C09159=1159.739,-99.599,-42.687,178.880,5.876,149.381
C09160=1159.744,-99.849,-42.678,178.877,5.876,149.382
C09161=1159.750,-100.100,-42.669,178.875,5.875,149.382
C09162=1159.755,-100.349,-42.659,178.874,5.875,149.383
C09163=1159.760,-100.599,-42.650,178.871,5.875,149.383
C09164=1159.766,-100.849,-42.641,178.869,5.875,149.384
C09165=1159.771,-101.098,-42.631,178.867,5.874,149.384
C09166=1159.777,-101.348,-42.622,178.864,5.874,149.385
C09167=1159.782,-101.598,-42.613,178.863,5.874,149.386
C09168=1159.787,-101.848,-42.604,178.861,5.873,149.386
C09169=1159.793,-102.120,-42.594,178.859,5.874,149.387
C09170=1159.799,-102.392,-42.583,178.856,5.873,149.387
C09171=1159.805,-102.664,-42.573,178.854,5.872,149.388
C09172=1159.810,-102.936,-42.562,178.852,5.872,149.389
C09173=1159.815,-103.186,-42.554,178.849,5.872,149.389
C09174=1159.821,-103.436,-42.544,178.847,5.871,149.390
C09175=1159.826,-103.686,-42.535,178.846,5.871,149.390
C09176=1159.831,-103.935,-42.526,178.843,5.871,149.391
C09177=1159.836,-104.185,-42.517,178.841,5.870,149.391
C09178=1159.842,-104.435,-42.507,178.839,5.870,149.392
C09179=1159.847,-104.685,-42.498,178.837,5.870,149.393
C09180=1159.853,-104.933,-42.489,178.835,5.870,149.393
C09181=1159.859,-105.184,-42.479,178.833,5.869,149.394
C09182=1159.864,-105.433,-42.471,178.831,5.870,149.394
C09183=1159.869,-105.683,-42.462,178.828,5.869,149.395
C09184=1159.874,-105.933,-42.453,178.826,5.868,149.395
C09185=1159.880,-106.183,-42.443,178.825,5.868,149.396
C09186=1159.885,-106.432,-42.434,178.822,5.868,149.396
C09187=1159.890,-106.682,-42.425,178.820,5.868,149.397
C09188=1159.895,-106.932,-42.416,178.818,5.867,149.397
C09189=1159.901,-107.182,-42.406,178.816,5.867,149.398
C09190=1159.906,-107.432,-42.397,178.814,5.867,149.399
C09191=1159.911,-107.681,-42.388,178.812,5.866,149.399
C09192=1159.917,-107.931,-42.379,178.810,5.866,149.400
C09193=1159.922,-108.181,-42.369,178.807,5.865,149.400
C09194=1159.928,-108.431,-42.361,178.806,5.865,149.401
C09195=1159.933,-108.680,-42.352,178.804,5.865,149.401
C09196=1159.939,-108.930,-42.343,178.802,5.865,149.402
C09197=1159.944,-109.180,-42.334,178.799,5.864,149.403
C09198=1159.949,-109.430,-42.324,178.797,5.864,149.403
C09199=1159.954,-109.680,-42.315,178.795,5.864,149.404
C09200=1159.960,-109.929,-42.306,178.793,5.863,149.404
C09201=1159.965,-110.179,-42.297,178.791,5.863,149.405
C09202=1159.970,-110.429,-42.288,178.789,5.863,149.405
C09203=1159.976,-110.679,-42.279,178.787,5.863,149.406
C09204=1159.982,-110.928,-42.270,178.785,5.862,149.406
C09205=1159.987,-111.178,-42.262,178.783,5.862,149.407
C09206=1159.992,-111.428,-42.253,178.781,5.862,149.408
C09207=1159.997,-111.678,-42.244,178.778,5.861,149.408
C09208=1160.002,-111.928,-42.235,178.777,5.861,149.409
C09209=1160.008,-112.178,-42.225,178.775,5.860,149.409
C09210=1160.013,-112.428,-42.216,178.773,5.861,149.410
C09211=1160.019,-112.678,-42.208,178.770,5.860,149.410
C09212=1160.024,-112.927,-42.199,178.769,5.860,149.411
C09213=1160.029,-113.177,-42.190,178.767,5.859,149.411
C09214=1160.035,-113.427,-42.181,178.764,5.860,149.412
C09215=1160.040,-113.676,-42.172,178.762,5.859,149.412
C09216=1160.045,-113.926,-42.163,178.761,5.859,149.413
C09217=1160.051,-114.176,-42.154,178.758,5.858,149.413
C09218=1160.057,-114.426,-42.145,178.756,5.858,149.414
C09219=1160.062,-114.675,-42.137,178.754,5.858,149.415
C09220=1160.067,-114.925,-42.128,178.752,5.857,149.415
C09221=1160.072,-115.175,-42.119,178.750,5.857,149.416
C09222=1160.077,-115.425,-42.110,178.748,5.857,149.416
C09223=1160.082,-115.675,-42.101,178.746,5.857,149.417
C09224=1160.088,-115.924,-42.092,178.744,5.856,149.417
C09225=1160.093,-116.174,-42.083,178.742,5.857,149.418
C09226=1160.099,-116.424,-42.075,178.740,5.856,149.418
C09227=1160.104,-116.674,-42.065,178.738,5.856,149.419
C09228=1160.110,-116.924,-42.056,178.736,5.855,149.419
C09229=1160.115,-117.173,-42.048,178.734,5.855,149.420
C09230=1160.121,-117.423,-42.039,178.732,5.855,149.421
C09231=1160.126,-117.673,-42.031,178.730,5.855,149.421
C09232=1160.131,-117.923,-42.022,178.728,5.854,149.422
C09233=1160.136,-118.173,-42.013,178.726,5.853,149.422
C09234=1160.142,-118.422,-42.004,178.724,5.854,149.423
C09235=1160.147,-118.672,-41.995,178.721,5.853,149.423
C09236=1160.152,-118.922,-41.986,178.720,5.853,149.424
C09237=1160.158,-119.172,-41.978,178.718,5.852,149.424
C09238=1160.164,-119.421,-41.970,178.715,5.853,149.425
C09239=1160.169,-119.671,-41.961,178.713,5.852,149.425
C09240=1160.174,-119.921,-41.952,178.712,5.852,149.426
C09241=1160.179,-120.171,-41.943,178.709,5.851,149.426
C09242=1160.185,-120.420,-41.935,178.707,5.852,149.427
C09243=1160.190,-120.670,-41.926,178.705,5.851,149.428
C09244=1160.196,-120.920,-41.917,178.704,5.851,149.428
C09245=1160.201,-121.170,-41.909,178.701,5.850,149.429
C09246=1160.207,-121.419,-41.900,178.699,5.851,149.429
C09247=1160.212,-121.669,-41.891,178.697,5.850,149.430
C09248=1160.217,-121.919,-41.882,178.696,5.850,149.430
C09249=1160.222,-122.169,-41.874,178.693,5.849,149.431
C09250=1160.228,-122.419,-41.866,178.692,5.849,149.431
C09251=1160.233,-122.668,-41.857,178.689,5.849,149.432
C09252=1160.238,-122.918,-41.848,178.687,5.849,149.432
C09253=1160.244,-123.169,-41.840,178.685,5.848,149.433
C09254=1160.250,-123.418,-41.831,178.684,5.848,149.433
C09255=1160.254,-123.668,-41.823,178.681,5.847,149.434
C09256=1160.259,-123.917,-41.814,178.679,5.848,149.435
C09257=1160.265,-124.168,-41.806,178.677,5.847,149.435
C09258=1160.271,-124.417,-41.797,178.676,5.847,149.436
C09259=1160.276,-124.667,-41.788,178.673,5.846,149.436
C09260=1160.281,-124.917,-41.780,178.671,5.847,149.437
C09261=1160.287,-125.166,-41.771,178.669,5.846,149.437
C09262=1160.292,-125.416,-41.763,178.668,5.846,149.438
C09263=1160.297,-125.666,-41.754,178.665,5.845,149.438
C09264=1160.303,-125.916,-41.746,178.664,5.845,149.439
C09265=1160.309,-126.166,-41.737,178.661,5.845,149.439
C09266=1160.313,-126.415,-41.729,178.659,5.845,149.440
C09267=1160.319,-126.665,-41.721,178.657,5.844,149.440
C09268=1160.324,-126.915,-41.712,178.656,5.844,149.441
C09269=1160.329,-127.165,-41.703,178.653,5.843,149.441
C09270=1160.335,-127.415,-41.695,178.651,5.844,149.442
C09271=1160.341,-127.664,-41.686,178.649,5.843,149.443
C09272=1160.346,-127.915,-41.678,178.648,5.843,149.443
C09273=1159.925,-127.926,-41.720,178.644,5.846,149.445
C09274=1159.919,-127.675,-41.728,178.645,5.846,149.444
C09275=1159.914,-127.425,-41.737,178.648,5.847,149.444
C09276=1159.908,-127.176,-41.745,178.650,5.847,149.443
C09277=1159.903,-126.926,-41.753,178.652,5.847,149.443
C09278=1159.898,-126.676,-41.762,178.653,5.847,149.442
C09279=1159.892,-126.427,-41.771,178.656,5.848,149.442
C09280=1159.887,-126.177,-41.779,178.658,5.848,149.441
C09281=1159.882,-125.927,-41.788,178.660,5.848,149.441
C09282=1159.876,-125.678,-41.796,178.661,5.848,149.440
C09283=1159.871,-125.427,-41.804,178.664,5.849,149.440
C09284=1159.865,-125.177,-41.813,178.665,5.849,149.439
C09285=1159.860,-124.927,-41.822,178.668,5.849,149.438
C09286=1159.855,-124.679,-41.830,178.670,5.849,149.438
C09287=1159.850,-124.428,-41.838,178.672,5.850,149.437
C09288=1159.845,-124.178,-41.847,178.673,5.850,149.437
C09289=1159.839,-123.929,-41.856,178.676,5.851,149.436
C09290=1159.833,-123.679,-41.864,178.678,5.851,149.436
C09291=1159.828,-123.429,-41.873,178.680,5.851,149.435
C09292=1159.822,-123.180,-41.881,178.681,5.851,149.435
C09293=1159.817,-122.930,-41.890,178.684,5.852,149.434
C09294=1159.812,-122.679,-41.898,178.685,5.852,149.434
C09295=1159.807,-122.430,-41.907,178.688,5.852,149.433
C09296=1159.801,-122.180,-41.916,178.690,5.853,149.433
C09297=1159.796,-121.931,-41.925,178.692,5.853,149.432
C09298=1159.790,-121.680,-41.933,178.694,5.854,149.432
C09299=1159.785,-121.430,-41.942,178.696,5.853,149.431
C09300=1159.779,-121.181,-41.950,178.698,5.854,149.430
C09301=1159.774,-120.931,-41.959,178.700,5.854,149.430
C09302=1159.769,-120.681,-41.968,178.702,5.855,149.429
C09303=1159.764,-120.432,-41.977,178.704,5.855,149.429
C09304=1159.758,-120.182,-41.985,178.706,5.855,149.428
C09305=1159.752,-119.932,-41.994,178.708,5.855,149.428
C09306=1159.747,-119.682,-42.003,178.710,5.856,149.427
C09307=1159.742,-119.432,-42.011,178.712,5.856,149.427
C09308=1159.736,-119.183,-42.020,178.714,5.856,149.426
C09309=1159.731,-118.933,-42.029,178.716,5.856,149.426
C09310=1159.726,-118.683,-42.037,178.718,5.857,149.425
C09311=1159.721,-118.433,-42.046,178.720,5.857,149.425
C09312=1159.715,-118.183,-42.055,178.722,5.858,149.424
C09313=1159.710,-117.934,-42.063,178.724,5.857,149.423
C09314=1159.704,-117.684,-42.072,178.726,5.858,149.423
C09315=1159.699,-117.434,-42.081,178.728,5.858,149.422
C09316=1159.694,-117.184,-42.090,178.730,5.859,149.422
C09317=1159.689,-116.934,-42.099,178.732,5.858,149.421
C09318=1159.683,-116.685,-42.107,178.734,5.859,149.421
C09319=1159.678,-116.435,-42.116,178.736,5.860,149.420
C09320=1159.673,-116.185,-42.125,178.738,5.860,149.420
C09321=1159.667,-115.935,-42.134,178.741,5.860,149.419
C09322=1159.662,-115.685,-42.142,178.742,5.860,149.419
C09323=1159.656,-115.436,-42.151,178.744,5.861,149.418
C09324=1159.651,-115.186,-42.160,178.746,5.861,149.418
C09325=1159.645,-114.936,-42.169,178.749,5.861,149.417
C09326=1159.640,-114.686,-42.178,178.750,5.861,149.416
C09327=1159.635,-114.436,-42.187,178.753,5.862,149.416
C09328=1159.629,-114.187,-42.196,178.754,5.862,149.415
C09329=1159.624,-113.937,-42.205,178.757,5.862,149.415
C09330=1159.619,-113.688,-42.213,178.758,5.862,149.414
C09331=1159.614,-113.438,-42.222,178.761,5.863,149.414
C09332=1159.609,-113.188,-42.231,178.763,5.864,149.413
C09333=1159.603,-112.938,-42.241,178.765,5.863,149.413
C09334=1159.597,-112.689,-42.249,178.767,5.864,149.412
C09335=1159.592,-112.439,-42.258,178.769,5.864,149.412
C09336=1159.587,-112.189,-42.267,178.771,5.864,149.411
C09337=1159.581,-111.939,-42.276,178.773,5.864,149.410
C09338=1159.576,-111.689,-42.285,178.775,5.865,149.410
C09339=1159.571,-111.439,-42.294,178.777,5.865,149.409
C09340=1159.565,-111.189,-42.303,178.779,5.865,149.409
C09341=1159.560,-110.939,-42.312,178.781,5.865,149.408
C09342=1159.554,-110.690,-42.321,178.783,5.866,149.408
C09343=1159.549,-110.440,-42.330,178.785,5.867,149.407
C09344=1159.544,-110.190,-42.339,178.787,5.867,149.407
C09345=1159.539,-109.941,-42.347,178.790,5.867,149.406
C09346=1159.533,-109.690,-42.357,178.791,5.867,149.406
C09347=1159.528,-109.441,-42.366,178.794,5.868,149.405
C09348=1159.523,-109.191,-42.375,178.796,5.868,149.404
C09349=1159.518,-108.941,-42.384,178.798,5.868,149.404
C09350=1159.513,-108.692,-42.393,178.799,5.868,149.403
C09351=1159.506,-108.442,-42.402,178.802,5.869,149.403
C09352=1159.501,-108.192,-42.411,178.804,5.869,149.402
C09353=1159.496,-107.942,-42.420,178.806,5.869,149.402
C09354=1159.491,-107.693,-42.429,178.808,5.870,149.401
C09355=1159.485,-107.442,-42.439,178.810,5.870,149.400
C09356=1159.480,-107.193,-42.448,178.812,5.871,149.400
C09357=1159.475,-106.943,-42.457,178.814,5.871,149.400
C09358=1159.469,-106.694,-42.466,178.817,5.871,149.399
C09359=1159.464,-106.443,-42.475,178.819,5.872,149.398
C09360=1159.458,-106.193,-42.484,178.820,5.872,149.398
C09361=1159.453,-105.944,-42.493,178.823,5.872,149.397
C09362=1159.448,-105.694,-42.503,178.825,5.872,149.397
C09363=1159.442,-105.444,-42.512,178.827,5.873,149.396
C09364=1159.437,-105.195,-42.521,178.829,5.872,149.395
C09365=1159.432,-104.945,-42.530,178.831,5.873,149.395
C09366=1159.426,-104.695,-42.539,178.833,5.874,149.394
C09367=1159.421,-104.446,-42.549,178.835,5.874,149.394
C09368=1159.416,-104.196,-42.558,178.838,5.874,149.393
C09369=1159.410,-103.946,-42.567,178.839,5.874,149.393
C09370=1159.405,-103.696,-42.576,178.841,5.875,149.392
C09371=1159.400,-103.447,-42.586,178.844,5.875,149.392
C09372=1159.394,-103.197,-42.595,178.846,5.875,149.391
C09373=1159.389,-102.947,-42.604,178.848,5.876,149.391
C09374=1159.383,-102.675,-42.614,178.850,5.876,149.390
C09375=1159.378,-102.403,-42.625,178.852,5.876,149.389
C09376=1159.372,-102.131,-42.635,178.855,5.877,149.389
C09377=1159.366,-101.859,-42.644,178.857,5.878,149.388
C09378=1159.361,-101.610,-42.654,178.859,5.877,149.387
C09379=1159.355,-101.360,-42.663,178.861,5.878,149.387
C09380=1159.350,-101.110,-42.672,178.863,5.878,149.387
C09381=1159.345,-100.861,-42.682,178.866,5.878,149.386
C09382=1159.339,-100.610,-42.691,178.868,5.879,149.385
C09383=1159.334,-100.360,-42.700,178.869,5.879,149.385
C09384=1159.329,-100.110,-42.711,178.872,5.879,149.384
C09385=1159.324,-99.861,-42.719,178.874,5.879,149.384
C09386=1159.318,-99.611,-42.728,178.876,5.880,149.383
C09387=1159.313,-99.361,-42.739,178.878,5.880,149.382
C09388=1159.308,-99.111,-42.747,178.880,5.880,149.382
C09389=1159.302,-98.861,-42.757,178.882,5.881,149.381
C09390=1159.297,-98.612,-42.767,178.884,5.881,149.381
C09391=1159.292,-98.362,-42.775,178.886,5.882,149.380
C09392=1159.286,-98.113,-42.786,178.889,5.882,149.380
C09393=1159.281,-97.863,-42.795,178.891,5.882,149.379
C09394=1159.275,-97.612,-42.804,178.893,5.883,149.379
C09395=1159.270,-97.363,-42.814,178.895,5.883,149.378
C09396=1159.265,-97.113,-42.823,178.897,5.883,149.377
C09397=1159.260,-96.864,-42.833,178.899,5.884,149.377
C09398=1159.254,-96.614,-42.842,178.901,5.884,149.376
C09399=1159.248,-96.364,-42.851,178.904,5.884,149.376
C09400=1159.244,-96.115,-42.861,178.905,5.884,149.375
C09401=1159.238,-95.864,-42.870,178.907,5.885,149.375
C09402=1159.233,-95.615,-42.880,178.910,5.885,149.374
C09403=1159.227,-95.365,-42.889,178.912,5.885,149.374
C09404=1159.222,-95.116,-42.899,178.914,5.886,149.373
C09405=1159.216,-94.866,-42.909,178.917,5.886,149.372
C09406=1159.212,-94.616,-42.918,178.918,5.886,149.372
C09407=1159.206,-94.366,-42.928,178.920,5.887,149.371
C09408=1159.201,-94.116,-42.938,178.922,5.887,149.371
C09409=1159.195,-93.866,-42.947,178.925,5.887,149.370
C09410=1159.190,-93.617,-42.957,178.927,5.888,149.370
C09411=1159.184,-93.367,-42.966,178.929,5.888,149.369
C09412=1159.180,-93.118,-42.976,178.931,5.889,149.369
C09413=1159.174,-92.867,-42.985,178.933,5.889,149.368
C09414=1159.169,-92.618,-42.995,178.935,5.889,149.367
C09415=1159.163,-92.368,-43.004,178.938,5.890,149.367
C09416=1159.159,-92.118,-43.014,178.940,5.889,149.366
C09417=1159.153,-91.868,-43.024,178.942,5.890,149.366
C09418=1159.148,-91.619,-43.033,178.944,5.891,149.365
C09419=1159.142,-91.369,-43.044,178.946,5.890,149.364
C09420=1159.137,-91.119,-43.053,178.948,5.891,149.364
C09421=1159.132,-90.870,-43.063,178.951,5.892,149.363
C09422=1159.126,-90.620,-43.072,178.953,5.892,149.363
C09423=1159.121,-90.370,-43.082,178.955,5.892,149.362
C09424=1159.116,-90.120,-43.091,178.957,5.893,149.362
C09425=1159.111,-89.870,-43.101,178.959,5.893,149.361
C09426=1159.105,-89.621,-43.112,178.961,5.893,149.361
C09427=1159.100,-89.371,-43.120,178.963,5.893,149.360
C09428=1159.094,-89.121,-43.131,178.966,5.894,149.359
C09429=1159.089,-88.872,-43.140,178.968,5.895,149.359
C09430=1159.084,-88.621,-43.150,178.970,5.894,149.358
C09431=1159.078,-88.372,-43.160,178.972,5.895,149.358
C09432=1159.074,-88.122,-43.170,178.974,5.896,149.357
C09433=1159.068,-87.872,-43.179,178.976,5.895,149.357
C09434=1159.063,-87.623,-43.189,178.978,5.896,149.356
C09435=1159.057,-87.374,-43.199,178.981,5.897,149.356
C09436=1159.052,-87.123,-43.209,178.983,5.896,149.355
C09437=1159.047,-86.873,-43.219,178.985,5.897,149.354
C09438=1159.041,-86.624,-43.229,178.988,5.898,149.354
C09439=1159.036,-86.374,-43.238,178.989,5.898,149.353
C09440=1159.031,-86.124,-43.248,178.991,5.898,149.353
C09441=1159.026,-85.874,-43.259,178.994,5.899,149.352
C09442=1159.021,-85.625,-43.268,178.996,5.899,149.352
C09443=1159.015,-85.375,-43.278,178.998,5.899,149.351
C09444=1159.009,-85.125,-43.288,179.001,5.900,149.350
C09445=1159.005,-84.875,-43.298,179.002,5.900,149.350
C09446=1159.000,-84.626,-43.308,179.005,5.900,149.349
C09447=1158.994,-84.376,-43.318,179.007,5.901,149.349
C09448=1158.989,-84.126,-43.327,179.009,5.901,149.348
C09449=1158.983,-83.877,-43.337,179.011,5.901,149.347
C09450=1158.978,-83.627,-43.348,179.013,5.902,149.347
C09451=1158.973,-83.377,-43.357,179.016,5.902,149.346
C09452=1158.967,-83.127,-43.367,179.018,5.902,149.346
C09453=1158.962,-82.878,-43.377,179.020,5.903,149.345
C09454=1158.957,-82.627,-43.388,179.022,5.903,149.345
C09455=1158.952,-82.378,-43.398,179.024,5.904,149.344
C09456=1158.946,-82.128,-43.407,179.027,5.904,149.343
C09457=1158.940,-81.879,-43.417,179.028,5.904,149.343
C09458=1158.936,-81.629,-43.427,179.031,5.905,149.342
C09459=1158.931,-81.379,-43.437,179.033,5.905,149.342
C09460=1158.925,-81.129,-43.448,179.035,5.905,149.341
C09461=1158.919,-80.880,-43.458,179.038,5.906,149.341
C09462=1158.915,-80.630,-43.468,179.040,5.906,149.340
C09463=1158.909,-80.380,-43.477,179.041,5.906,149.340
C09464=1158.904,-80.130,-43.488,179.044,5.907,149.339
C09465=1158.899,-79.880,-43.498,179.046,5.907,149.338
C09466=1158.893,-79.631,-43.508,179.048,5.907,149.338
C09467=1158.888,-79.381,-43.518,179.050,5.908,149.337
C09468=1158.883,-79.132,-43.528,179.053,5.909,149.337
C09469=1158.878,-78.881,-43.539,179.055,5.909,149.336
C09470=1158.872,-78.632,-43.549,179.057,5.909,149.336
C09471=1158.867,-78.383,-43.559,179.060,5.909,149.335
C09472=1158.862,-78.132,-43.569,179.062,5.910,149.334
C09473=1158.857,-77.883,-43.579,179.063,5.910,149.334
C09474=1158.851,-77.633,-43.589,179.066,5.910,149.333
C09475=1158.845,-77.383,-43.599,179.068,5.911,149.333
C09476=1158.840,-77.133,-43.610,179.070,5.911,149.332
C09477=1158.835,-76.884,-43.619,179.073,5.912,149.331
C09478=1158.829,-76.612,-43.631,179.075,5.912,149.331
C09479=1158.823,-76.342,-43.641,179.077,5.913,149.330
C09480=1158.818,-76.070,-43.653,179.080,5.913,149.330
C09481=1158.812,-75.798,-43.664,179.082,5.913,149.329
C09482=1158.807,-75.549,-43.674,179.084,5.914,149.328
C09483=1158.802,-75.299,-43.685,179.087,5.914,149.328
C09484=1158.796,-75.049,-43.695,179.089,5.915,149.327
C09485=1158.791,-74.800,-43.705,179.091,5.915,149.327
C09486=1158.786,-74.550,-43.716,179.093,5.915,149.326
C09487=1158.780,-74.300,-43.726,179.096,5.916,149.325
C09488=1158.774,-74.050,-43.736,179.097,5.916,149.325
C09489=1158.770,-73.801,-43.747,179.100,5.916,149.324
C09490=1158.765,-73.552,-43.757,179.102,5.917,149.324
C09491=1158.759,-73.302,-43.767,179.105,5.917,149.323
C09492=1158.754,-73.052,-43.778,179.106,5.917,149.323
C09493=1158.749,-72.802,-43.788,179.109,5.918,149.322
C09494=1158.743,-72.553,-43.798,179.111,5.919,149.321
C09495=1158.738,-72.302,-43.809,179.113,5.919,149.321
C09496=1158.732,-72.053,-43.819,179.115,5.919,149.320
C09497=1158.727,-71.803,-43.829,179.118,5.920,149.320
C09498=1158.722,-71.553,-43.840,179.120,5.920,149.319
C09499=1158.716,-71.304,-43.850,179.122,5.920,149.319
C09500=1158.712,-71.054,-43.861,179.125,5.920,149.318
C09501=1158.706,-70.804,-43.871,179.127,5.921,149.317
C09502=1158.701,-70.554,-43.882,179.129,5.922,149.317
C09503=1158.695,-70.305,-43.892,179.131,5.922,149.316
C09504=1158.690,-70.055,-43.902,179.133,5.922,149.316
C09505=1158.685,-69.805,-43.913,179.136,5.923,149.315
C09506=1158.679,-69.556,-43.924,179.138,5.923,149.315
C09507=1158.674,-69.306,-43.934,179.140,5.923,149.314
C09508=1158.669,-69.056,-43.945,179.142,5.924,149.313
C09509=1158.664,-68.806,-43.955,179.145,5.925,149.313
C09510=1158.658,-68.556,-43.965,179.147,5.924,149.312
C09511=1158.653,-68.307,-43.976,179.149,5.925,149.312
C09512=1158.648,-68.057,-43.987,179.152,5.926,149.311
C09513=1158.642,-67.808,-43.997,179.154,5.926,149.310
C09514=1158.637,-67.557,-44.008,179.156,5.926,149.310
C09515=1158.632,-67.308,-44.018,179.158,5.927,149.309
C09516=1158.627,-67.058,-44.029,179.161,5.927,149.309
C09517=1158.621,-66.809,-44.039,179.163,5.928,149.308
C09518=1158.616,-66.558,-44.050,179.164,5.928,149.308
C09519=1158.611,-66.310,-44.061,179.167,5.928,149.307
C09520=1158.606,-66.059,-44.072,179.169,5.929,149.306
C09521=1158.601,-65.810,-44.082,179.172,5.929,149.306
C09522=1158.596,-65.559,-44.092,179.174,5.929,149.305
C09523=1158.590,-65.311,-44.103,179.176,5.930,149.305
C09524=1158.585,-65.060,-44.114,179.178,5.931,149.304
C09525=1158.580,-64.811,-44.124,179.181,5.931,149.303
C09526=1158.575,-64.561,-44.135,179.183,5.931,149.303
C09527=1158.569,-64.312,-44.145,179.185,5.932,149.302
C09528=1158.564,-64.061,-44.156,179.188,5.932,149.302
C09529=1158.558,-63.812,-44.168,179.190,5.933,149.301
C09530=1158.553,-63.562,-44.178,179.192,5.933,149.301
C09531=1158.548,-63.312,-44.188,179.194,5.933,149.300
C09532=1158.543,-63.063,-44.200,179.197,5.934,149.299
C09533=1158.537,-62.813,-44.210,179.199,5.935,149.299
C09534=1158.532,-62.563,-44.220,179.201,5.935,149.298
C09535=1158.527,-62.314,-44.231,179.203,5.935,149.298
C09536=1158.522,-62.064,-44.242,179.206,5.935,149.297
C09537=1158.516,-61.815,-44.253,179.208,5.936,149.296
C09538=1158.511,-61.564,-44.264,179.210,5.937,149.296
C09539=1158.506,-61.315,-44.275,179.212,5.937,149.295
C09540=1158.501,-61.065,-44.286,179.214,5.937,149.295
C09541=1158.495,-60.816,-44.296,179.217,5.938,149.294
C09542=1158.491,-60.566,-44.307,179.219,5.938,149.294
C09543=1158.486,-60.316,-44.318,179.221,5.938,149.293
C09544=1158.480,-60.066,-44.329,179.223,5.939,149.292
C09545=1158.475,-59.816,-44.340,179.226,5.939,149.292
C09546=1158.469,-59.567,-44.351,179.228,5.940,149.291
C09547=1158.464,-59.317,-44.361,179.231,5.940,149.291
C09548=1158.459,-59.068,-44.372,179.233,5.940,149.290
C09549=1158.453,-58.818,-44.383,179.235,5.941,149.289
C09550=1158.449,-58.568,-44.395,179.237,5.942,149.289
C09551=1158.443,-58.318,-44.405,179.240,5.942,149.288
C09552=1158.438,-58.069,-44.416,179.242,5.943,149.288
C09553=1158.433,-57.819,-44.426,179.244,5.943,149.287
C09554=1158.427,-57.569,-44.438,179.247,5.943,149.287
C09555=1158.422,-57.319,-44.449,179.249,5.944,149.286
C09556=1158.417,-57.070,-44.460,179.251,5.944,149.285
C09557=1158.412,-56.820,-44.470,179.254,5.945,149.285
C09558=1158.406,-56.571,-44.482,179.256,5.945,149.284
C09559=1158.401,-56.320,-44.492,179.258,5.946,149.284
C09560=1158.396,-56.071,-44.504,179.261,5.946,149.283
C09561=1158.391,-55.822,-44.515,179.263,5.947,149.283
C09562=1158.385,-55.571,-44.526,179.265,5.947,149.282
C09563=1158.380,-55.322,-44.537,179.267,5.947,149.281
C09564=1158.375,-55.072,-44.547,179.270,5.948,149.281
C09565=1158.370,-54.822,-44.559,179.272,5.948,149.280
C09566=1158.364,-54.573,-44.570,179.274,5.949,149.280
C09567=1158.359,-54.323,-44.581,179.277,5.950,149.279
C09568=1158.354,-54.073,-44.592,179.278,5.950,149.279
C09569=1158.349,-53.824,-44.603,179.281,5.950,149.278
C09570=1158.343,-53.574,-44.614,179.283,5.951,149.277
C09571=1158.339,-53.324,-44.625,179.286,5.951,149.277
C09572=1158.333,-53.075,-44.635,179.288,5.952,149.276
C09573=1158.328,-52.825,-44.647,179.290,5.952,149.275
C09574=1158.323,-52.575,-44.659,179.292,5.952,149.275
C09575=1158.317,-52.326,-44.669,179.295,5.953,149.274
C09576=1158.312,-52.076,-44.681,179.297,5.954,149.274
C09577=1158.307,-51.826,-44.692,179.300,5.954,149.273
C09578=1158.302,-51.577,-44.703,179.302,5.955,149.273
C09579=1158.296,-51.327,-44.714,179.304,5.954,149.272
C09580=1158.292,-51.077,-44.725,179.306,5.955,149.271
C09581=1158.286,-50.828,-44.737,179.309,5.956,149.271
C09582=1158.281,-50.557,-44.749,179.311,5.956,149.270
C09583=1158.275,-50.286,-44.761,179.314,5.957,149.270
C09584=1158.269,-50.016,-44.773,179.316,5.957,149.269
C09585=1158.264,-49.745,-44.786,179.319,5.958,149.268
C09586=1158.259,-49.495,-44.796,179.321,5.958,149.268
C09587=1158.253,-49.246,-44.808,179.323,5.959,149.267
C09588=1158.248,-48.996,-44.819,179.326,5.959,149.266
C09589=1158.242,-48.746,-44.831,179.328,5.960,149.266
C09590=1158.237,-48.496,-44.842,179.330,5.960,149.265
C09591=1158.231,-48.247,-44.853,179.333,5.961,149.265
C09592=1158.227,-47.997,-44.864,179.335,5.961,149.264
C09593=1158.222,-47.748,-44.876,179.337,5.962,149.264
C09594=1158.216,-47.498,-44.887,179.340,5.962,149.263
C09595=1158.211,-47.249,-44.898,179.342,5.962,149.262
C09596=1158.206,-46.998,-44.910,179.344,5.963,149.262
C09597=1158.201,-46.749,-44.921,179.347,5.964,149.261
C09598=1158.195,-46.499,-44.932,179.349,5.964,149.261
C09599=1158.190,-46.250,-44.944,179.351,5.965,149.260
C09600=1158.185,-46.000,-44.956,179.354,5.965,149.259
C09601=1158.180,-45.750,-44.967,179.356,5.965,149.259
C09602=1158.174,-45.501,-44.978,179.358,5.966,149.258
C09603=1158.169,-45.251,-44.989,179.360,5.966,149.258
C09604=1158.164,-45.001,-45.001,179.363,5.967,149.257
C09605=1158.159,-44.751,-45.012,179.365,5.968,149.257
C09606=1158.153,-44.501,-45.024,179.368,5.968,149.256
C09607=1158.148,-44.252,-45.035,179.370,5.969,149.255
C09608=1158.143,-44.002,-45.047,179.372,5.968,149.255
C09609=1158.138,-43.753,-45.058,179.374,5.969,149.254
C09610=1158.133,-43.503,-45.070,179.377,5.970,149.254
C09611=1158.128,-43.253,-45.081,179.379,5.970,149.253
C09612=1158.122,-43.004,-45.093,179.382,5.971,149.252
C09613=1158.117,-42.754,-45.104,179.384,5.972,149.252
C09614=1158.112,-42.504,-45.116,179.387,5.972,149.251
C09615=1158.107,-42.255,-45.127,179.389,5.973,149.251
C09616=1158.102,-42.005,-45.139,179.391,5.972,149.250
C09617=1158.096,-41.756,-45.151,179.393,5.973,149.250
C09618=1158.091,-41.506,-45.162,179.396,5.974,149.249
C09619=1158.085,-41.256,-45.174,179.398,5.974,149.248
C09620=1158.081,-41.006,-45.185,179.401,5.975,149.248
C09621=1158.075,-40.756,-45.197,179.403,5.976,149.247
C09622=1158.071,-40.507,-45.208,179.406,5.976,149.246
C09623=1158.065,-40.258,-45.220,179.408,5.977,149.246
C09624=1158.059,-40.008,-45.232,179.410,5.976,149.245
C09625=1158.055,-39.758,-45.243,179.412,5.977,149.245
C09626=1158.049,-39.508,-45.255,179.415,5.978,149.244
C09627=1158.044,-39.258,-45.267,179.417,5.978,149.244
C09628=1158.039,-39.009,-45.278,179.420,5.979,149.243
C09629=1158.034,-38.759,-45.290,179.422,5.980,149.242
C09630=1158.028,-38.510,-45.302,179.424,5.980,149.242
C09631=1158.023,-38.260,-45.314,179.427,5.981,149.241
C09632=1158.018,-38.010,-45.325,179.429,5.981,149.241
C09633=1158.012,-37.760,-45.337,179.431,5.981,149.240
C09634=1158.008,-37.511,-45.349,179.434,5.982,149.239
C09635=1158.002,-37.261,-45.360,179.436,5.983,149.239
C09636=1157.997,-37.011,-45.372,179.438,5.983,149.238
C09637=1157.992,-36.761,-45.384,179.441,5.984,149.238
C09638=1157.987,-36.512,-45.396,179.443,5.984,149.237
C09639=1157.981,-36.263,-45.408,179.445,5.985,149.237
C09640=1157.976,-36.013,-45.419,179.448,5.985,149.236
C09641=1157.971,-35.763,-45.431,179.450,5.986,149.235
C09642=1157.965,-35.513,-45.443,179.453,5.987,149.235
C09643=1157.961,-35.264,-45.455,179.454,5.987,149.234
C09644=1157.955,-35.014,-45.467,179.457,5.987,149.234
C09645=1157.950,-34.764,-45.479,179.459,5.988,149.233
C09646=1157.945,-34.514,-45.490,179.462,5.988,149.232
C09647=1157.940,-34.265,-45.502,179.464,5.989,149.232
C09648=1157.935,-34.016,-45.514,179.467,5.989,149.231
C09649=1157.929,-33.766,-45.526,179.469,5.990,149.231
C09650=1157.924,-33.516,-45.538,179.472,5.991,149.230
C09651=1157.919,-33.266,-45.549,179.474,5.991,149.230
C09652=1157.914,-33.017,-45.562,179.477,5.992,149.229
C09653=1157.908,-32.767,-45.574,179.479,5.993,149.228
C09654=1157.903,-32.518,-45.585,179.481,5.993,149.228
C09655=1157.898,-32.269,-45.597,179.483,5.993,149.227
C09656=1157.893,-32.019,-45.609,179.486,5.994,149.227
C09657=1157.887,-31.769,-45.621,179.488,5.994,149.226
C09658=1157.882,-31.519,-45.634,179.490,5.995,149.225
C09659=1157.877,-31.269,-45.646,179.493,5.996,149.225
C09660=1157.872,-31.020,-45.657,179.495,5.996,149.224
C09661=1157.867,-30.770,-45.670,179.498,5.997,149.224
C09662=1157.862,-30.521,-45.681,179.500,5.997,149.223
C09663=1157.856,-30.271,-45.693,179.502,5.998,149.223
C09664=1157.851,-30.021,-45.706,179.505,5.998,149.222
C09665=1157.846,-29.771,-45.718,179.507,5.999,149.221
C09666=1157.841,-29.522,-45.729,179.510,6.000,149.221
C09667=1157.836,-29.272,-45.742,179.512,6.000,149.220
C09668=1157.830,-29.022,-45.754,179.515,6.001,149.219
C09669=1157.825,-28.773,-45.766,179.517,6.002,149.219
C09670=1157.820,-28.523,-45.778,179.519,6.001,149.218
C09671=1157.814,-28.273,-45.790,179.521,6.002,149.218
C09672=1157.809,-28.024,-45.803,179.524,6.003,149.217
C09673=1157.805,-27.774,-45.814,179.526,6.003,149.217
C09674=1157.799,-27.525,-45.826,179.529,6.004,149.216
C09675=1157.795,-27.274,-45.839,179.531,6.005,149.215
C09676=1157.790,-27.025,-45.851,179.533,6.005,149.215
C09677=1157.784,-26.775,-45.863,179.536,6.005,149.214
C09678=1157.779,-26.526,-45.876,179.538,6.006,149.214
C09679=1157.774,-26.276,-45.888,179.541,6.007,149.213
C09680=1157.768,-26.027,-45.900,179.543,6.007,149.212
C09681=1157.763,-25.777,-45.912,179.546,6.008,149.212
C09682=1157.758,-25.527,-45.925,179.548,6.009,149.211
C09683=1157.753,-25.278,-45.936,179.551,6.009,149.211
C09684=1157.748,-25.028,-45.949,179.553,6.010,149.210
C09685=1157.743,-24.778,-45.961,179.556,6.010,149.209
C09686=1157.737,-24.508,-45.975,179.558,6.011,149.209
C09687=1157.731,-24.239,-45.987,179.560,6.012,149.208
C09688=1157.726,-23.968,-46.000,179.563,6.012,149.208
C09689=1157.721,-23.699,-46.014,179.566,6.012,149.207
C09690=1157.715,-23.449,-46.026,179.568,6.013,149.206
C09691=1157.710,-23.199,-46.039,179.571,6.014,149.206
C09692=1157.705,-22.950,-46.051,179.573,6.014,149.205
C09693=1157.700,-22.700,-46.063,179.575,6.015,149.205
C09694=1157.694,-22.451,-46.076,179.578,6.016,149.204
C09695=1157.689,-22.201,-46.088,179.580,6.016,149.203
C09696=1157.684,-21.952,-46.100,179.582,6.017,149.203
C09697=1157.679,-21.702,-46.113,179.585,6.017,149.202
C09698=1157.674,-21.452,-46.125,179.587,6.018,149.202
C09699=1157.668,-21.202,-46.138,179.590,6.019,149.201
C09700=1157.663,-20.953,-46.151,179.592,6.019,149.201
C09701=1157.658,-20.703,-46.163,179.595,6.020,149.200
C09702=1157.652,-20.453,-46.175,179.597,6.021,149.199
C09703=1157.647,-20.204,-46.188,179.600,6.021,149.199
C09704=1157.642,-19.953,-46.200,179.602,6.022,149.198
C09705=1157.637,-19.704,-46.213,179.604,6.022,149.198
C09706=1157.632,-19.455,-46.225,179.607,6.023,149.197
C09707=1157.627,-19.205,-46.237,179.609,6.024,149.196
C09708=1157.622,-18.956,-46.250,179.611,6.024,149.196
C09709=1157.617,-18.706,-46.262,179.614,6.025,149.195
C09710=1157.612,-18.456,-46.275,179.616,6.026,149.195
C09711=1157.607,-18.206,-46.287,179.619,6.026,149.194
C09712=1157.601,-17.957,-46.300,179.621,6.027,149.194
C09713=1157.596,-17.707,-46.313,179.624,6.027,149.193
C09714=1157.590,-17.458,-46.326,179.626,6.028,149.192
C09715=1157.585,-17.208,-46.338,179.629,6.029,149.192
C09716=1157.580,-16.958,-46.351,179.631,6.029,149.191
C09717=1157.575,-16.709,-46.363,179.633,6.030,149.191
C09718=1157.570,-16.459,-46.376,179.636,6.030,149.190
C09719=1157.565,-16.210,-46.388,179.638,6.031,149.189
C09720=1157.559,-15.960,-46.401,179.641,6.031,149.189
C09721=1157.554,-15.710,-46.414,179.643,6.032,149.188
C09722=1157.549,-15.461,-46.426,179.646,6.033,149.188
C09723=1157.544,-15.211,-46.439,179.648,6.034,149.187
C09724=1157.539,-14.962,-46.452,179.651,6.034,149.186
C09725=1157.535,-14.712,-46.465,179.653,6.035,149.186
C09726=1157.529,-14.462,-46.478,179.655,6.035,149.185
C09727=1157.523,-14.212,-46.490,179.658,6.036,149.185
C09728=1157.518,-13.963,-46.502,179.660,6.036,149.184
C09729=1157.514,-13.713,-46.515,179.662,6.037,149.184
C09730=1157.508,-13.464,-46.528,179.665,6.038,149.183
C09731=1157.503,-13.214,-46.541,179.667,6.039,149.182
C09732=1157.497,-12.965,-46.554,179.670,6.039,149.182
C09733=1157.493,-12.715,-46.567,179.673,6.041,149.181
C09734=1157.488,-12.465,-46.579,179.675,6.041,149.181
C09735=1157.483,-12.216,-46.592,179.678,6.042,149.180
C09736=1157.477,-11.966,-46.605,179.680,6.042,149.179
C09737=1157.472,-11.716,-46.618,179.683,6.043,149.179
C09738=1157.467,-11.467,-46.631,179.685,6.043,149.178
C09739=1157.462,-11.218,-46.643,179.688,6.044,149.178
C09740=1157.457,-10.967,-46.657,179.690,6.045,149.177
C09741=1157.452,-10.718,-46.669,179.693,6.045,149.176
C09742=1157.447,-10.469,-46.682,179.695,6.046,149.176
C09743=1157.441,-10.218,-46.695,179.697,6.046,149.175
C09744=1157.436,-9.969,-46.708,179.700,6.047,149.175
C09745=1157.431,-9.720,-46.721,179.702,6.048,149.174
C09746=1157.426,-9.471,-46.733,179.704,6.048,149.174
C09747=1157.421,-9.220,-46.747,179.707,6.049,149.173
C09748=1157.416,-8.971,-46.759,179.709,6.050,149.172
C09749=1157.410,-8.722,-46.772,179.712,6.050,149.172
C09750=1157.405,-8.471,-46.786,179.714,6.051,149.171
C09751=1157.400,-8.222,-46.798,179.717,6.051,149.171
C09752=1157.395,-7.973,-46.811,179.719,6.052,149.170
C09753=1157.390,-7.722,-46.824,179.722,6.053,149.169
C09754=1157.385,-7.473,-46.837,179.724,6.054,149.169
C09755=1157.380,-7.223,-46.850,179.727,6.055,149.168
C09756=1157.374,-6.973,-46.863,179.729,6.056,149.168
C09757=1157.369,-6.725,-46.876,179.732,6.056,149.167
C09758=1157.365,-6.475,-46.889,179.734,6.056,149.166
C09759=1157.359,-6.225,-46.903,179.737,6.057,149.166
C09760=1157.354,-5.976,-46.915,179.739,6.058,149.165
C09761=1157.349,-5.725,-46.929,179.741,6.059,149.165
C09762=1157.343,-5.476,-46.941,179.744,6.059,149.164
C09763=1157.338,-5.227,-46.954,179.746,6.060,149.164
C09764=1157.333,-4.977,-46.968,179.749,6.060,149.163
C09765=1157.328,-4.728,-46.981,179.751,6.061,149.163
C09766=1157.323,-4.477,-46.994,179.754,6.061,149.162
C09767=1157.318,-4.228,-47.007,179.757,6.063,149.161
C09768=1157.313,-3.979,-47.020,179.759,6.064,149.161
C09769=1157.308,-3.729,-47.034,179.761,6.064,149.160
C09770=1157.303,-3.480,-47.046,179.764,6.065,149.160
C09771=1157.297,-3.229,-47.060,179.766,6.066,149.159
C09772=1157.292,-2.980,-47.073,179.769,6.066,149.158
C09773=1157.287,-2.730,-47.087,179.771,6.067,149.158
C09774=1157.282,-2.481,-47.100,179.774,6.067,149.157
C09775=1157.276,-2.231,-47.113,179.776,6.068,149.157
C09776=1157.272,-1.981,-47.126,179.779,6.069,149.156
C09777=1157.266,-1.732,-47.140,179.781,6.069,149.156
C09778=1157.262,-1.482,-47.153,179.784,6.071,149.155
C09779=1157.256,-1.233,-47.166,179.786,6.071,149.154
C09780=1157.252,-0.983,-47.179,179.789,6.072,149.154
C09781=1157.246,-0.734,-47.193,179.791,6.073,149.153
C09782=1157.241,-0.484,-47.205,179.794,6.073,149.153
C09783=1157.236,-0.235,-47.220,179.796,6.074,149.152
C09784=1157.231,0.015,-47.232,179.798,6.074,149.151
C09785=1157.225,0.265,-47.246,179.801,6.075,149.151
C09786=1157.221,0.514,-47.259,179.803,6.076,149.150
C09787=1157.215,0.764,-47.273,179.807,6.077,149.150
C09788=1157.210,1.013,-47.285,179.809,6.078,149.149
C09789=1157.205,1.263,-47.299,179.811,6.078,149.148
C09790=1157.199,1.532,-47.314,179.814,6.079,149.148
C09791=1157.194,1.802,-47.328,179.816,6.079,149.147
C09792=1157.189,2.071,-47.343,179.819,6.081,149.147
C09793=1157.183,2.341,-47.357,179.822,6.081,149.146
C09794=1157.177,2.590,-47.371,179.824,6.082,149.145
C09795=1157.173,2.840,-47.384,179.827,6.082,149.145
C09796=1157.167,3.089,-47.398,179.829,6.083,149.144
C09797=1157.163,3.339,-47.411,179.832,6.084,149.144
C09798=1157.157,3.588,-47.425,179.835,6.085,149.143
C09799=1157.152,3.838,-47.438,179.837,6.086,149.142
C09800=1157.147,4.087,-47.452,179.839,6.087,149.142
C09801=1157.142,4.337,-47.465,179.842,6.087,149.141
C09802=1157.137,4.586,-47.478,179.844,6.088,149.141
C09803=1157.132,4.836,-47.492,179.847,6.088,149.140
C09804=1157.126,5.085,-47.506,179.849,6.089,149.140
C09805=1157.122,5.335,-47.519,179.852,6.090,149.139
C09806=1157.117,5.585,-47.533,179.854,6.091,149.139
C09807=1157.111,5.835,-47.546,179.857,6.092,149.138
C09808=1157.107,6.084,-47.560,179.859,6.092,149.137
C09809=1157.101,6.334,-47.573,179.862,6.093,149.137
C09810=1157.096,6.584,-47.587,179.864,6.094,149.136
C09811=1157.091,6.832,-47.601,179.867,6.094,149.136
C09812=1157.086,7.083,-47.614,179.870,6.096,149.135
C09813=1157.081,7.332,-47.629,179.872,6.096,149.134
C09814=1157.075,7.582,-47.642,179.874,6.097,149.134
C09815=1157.071,7.831,-47.656,179.877,6.098,149.133
C09816=1157.065,8.080,-47.669,179.879,6.098,149.133
C09817=1157.060,8.331,-47.683,179.882,6.099,149.132
C09818=1157.056,8.580,-47.697,179.884,6.100,149.132
C09819=1157.050,8.829,-47.711,179.887,6.101,149.131
C09820=1157.045,9.079,-47.724,179.889,6.102,149.131
C09821=1157.039,9.328,-47.738,179.892,6.102,149.130
C09822=1157.035,9.578,-47.752,179.895,6.103,149.129
C09823=1157.030,9.828,-47.765,179.897,6.103,149.129
C09824=1157.024,10.077,-47.779,179.900,6.104,149.128
C09825=1157.019,10.327,-47.793,179.902,6.106,149.128
C09826=1157.014,10.577,-47.807,179.905,6.106,149.127
C09827=1157.009,10.826,-47.820,179.907,6.107,149.126
C09828=1157.004,11.076,-47.835,179.910,6.107,149.126
C09829=1156.999,11.325,-47.849,179.912,6.108,149.125
C09830=1156.994,11.575,-47.862,179.915,6.109,149.125
C09831=1156.989,11.825,-47.876,179.917,6.110,149.124
C09832=1156.984,12.073,-47.890,179.920,6.111,149.123
C09833=1156.979,12.323,-47.904,179.922,6.112,149.123
C09834=1156.974,12.573,-47.918,179.925,6.112,149.122
C09835=1156.968,12.822,-47.931,179.927,6.113,149.122
C09836=1156.963,13.072,-47.946,179.930,6.114,149.121
C09837=1156.958,13.322,-47.960,179.932,6.115,149.121
C09838=1156.954,13.571,-47.974,179.935,6.115,149.120
C09839=1156.948,13.821,-47.987,179.937,6.116,149.120
C09840=1156.943,14.071,-48.001,179.940,6.117,149.119
C09841=1156.938,14.320,-48.015,179.943,6.118,149.118
C09842=1156.933,14.569,-48.029,179.945,6.119,149.118
C09843=1156.928,14.819,-48.044,179.947,6.120,149.117
C09844=1156.923,15.069,-48.058,179.950,6.120,149.117
C09845=1156.917,15.318,-48.072,179.952,6.121,149.116
C09846=1156.913,15.568,-48.085,179.956,6.122,149.115
C09847=1156.908,15.817,-48.099,179.958,6.123,149.115
C09848=1156.903,16.067,-48.113,179.960,6.123,149.114
C09849=1156.897,16.316,-48.127,179.963,6.124,149.114
C09850=1156.892,16.566,-48.142,179.965,6.125,149.113
C09851=1156.887,16.816,-48.156,179.968,6.126,149.113
C09852=1156.882,17.065,-48.170,179.971,6.127,149.112
C09853=1156.877,17.314,-48.184,179.973,6.128,149.112
C09854=1156.872,17.564,-48.198,179.975,6.128,149.111
C09855=1156.867,17.814,-48.213,179.978,6.129,149.110
C09856=1156.862,18.063,-48.227,179.981,6.130,149.110
C09857=1156.856,18.312,-48.241,179.983,6.131,149.109
C09858=1156.851,18.562,-48.255,179.986,6.131,149.109
C09859=1156.846,18.812,-48.269,179.988,6.132,149.108
C09860=1156.841,19.062,-48.284,179.991,6.134,149.107
C09861=1156.836,19.311,-48.297,179.993,6.134,149.107
C09862=1156.831,19.560,-48.312,179.996,6.135,149.106
C09863=1156.826,19.810,-48.326,179.998,6.136,149.106
C09864=1156.821,20.060,-48.340,-179.999,6.136,149.105
C09865=1156.816,20.309,-48.355,-179.997,6.138,149.105
C09866=1156.810,20.558,-48.369,-179.994,6.138,149.104
C09867=1156.806,20.808,-48.383,-179.992,6.139,149.104
C09868=1156.801,21.058,-48.397,-179.989,6.139,149.103
C09869=1156.796,21.308,-48.411,-179.986,6.141,149.102
C09870=1156.791,21.557,-48.426,-179.984,6.142,149.102
C09871=1156.785,21.806,-48.440,-179.982,6.142,149.101
C09872=1156.780,22.055,-48.455,-179.979,6.143,149.101
C09873=1156.775,22.305,-48.469,-179.976,6.145,149.100
C09874=1156.771,22.555,-48.483,-179.973,6.145,149.100
C09875=1156.766,22.804,-48.497,-179.971,6.146,149.099
C09876=1156.761,23.054,-48.512,-179.969,6.146,149.098
C09877=1156.754,23.303,-48.526,-179.966,6.148,149.098
C09878=1156.749,23.553,-48.540,-179.963,6.148,149.097
C09879=1156.745,23.802,-48.555,-179.961,6.149,149.097
C09880=1156.740,24.052,-48.570,-179.958,6.150,149.096
C09881=1156.735,24.302,-48.584,-179.956,6.151,149.096
C09882=1156.730,24.551,-48.598,-179.953,6.152,149.095
C09883=1156.725,24.801,-48.613,-179.951,6.153,149.095
C09884=1156.720,25.050,-48.627,-179.948,6.153,149.094
C09885=1156.714,25.300,-48.642,-179.945,6.155,149.093
C09886=1156.709,25.549,-48.656,-179.943,6.155,149.093
C09887=1156.704,25.799,-48.671,-179.941,6.156,149.092
C09888=1156.699,26.048,-48.686,-179.937,6.157,149.092
C09889=1156.694,26.298,-48.700,-179.935,6.158,149.091
C09890=1156.689,26.547,-48.714,-179.933,6.159,149.090
C09891=1156.684,26.798,-48.729,-179.930,6.159,149.090
C09892=1156.679,27.047,-48.744,-179.927,6.161,149.089
C09893=1156.674,27.296,-48.758,-179.925,6.162,149.089
C09894=1156.668,27.564,-48.774,-179.922,6.162,149.088
C09895=1156.663,27.834,-48.790,-179.919,6.163,149.088
C09896=1156.657,28.102,-48.806,-179.917,6.164,149.087
C09897=1156.652,28.372,-48.821,-179.914,6.165,149.086
C09898=1156.647,28.621,-48.836,-179.912,6.166,149.086
C09899=1156.642,28.871,-48.850,-179.909,6.167,149.085
C09900=1156.637,29.121,-48.865,-179.906,6.168,149.085
C09901=1156.632,29.370,-48.880,-179.904,6.169,149.084
C09902=1156.627,29.619,-48.894,-179.901,6.170,149.084
C09903=1156.622,29.869,-48.910,-179.899,6.170,149.083
C09904=1156.617,30.118,-48.924,-179.896,6.172,149.083
C09905=1156.612,30.368,-48.938,-179.893,6.172,149.082
C09906=1156.607,30.617,-48.953,-179.891,6.173,149.081
C09907=1156.602,30.867,-48.968,-179.888,6.174,149.081
C09908=1156.597,31.116,-48.983,-179.886,6.175,149.080
C09909=1156.592,31.366,-48.997,-179.883,6.176,149.080
C09910=1156.587,31.615,-49.013,-179.880,6.177,149.079
C09911=1156.582,31.865,-49.027,-179.878,6.178,149.078
C09912=1156.577,32.114,-49.042,-179.876,6.179,149.078
C09913=1156.571,32.364,-49.057,-179.873,6.179,149.077
C09914=1156.567,32.613,-49.072,-179.870,6.181,149.077
C09915=1156.562,32.863,-49.086,-179.867,6.181,149.076
C09916=1156.556,33.113,-49.102,-179.865,6.182,149.076
C09917=1156.551,33.362,-49.116,-179.862,6.183,149.075
C09918=1156.547,33.611,-49.131,-179.860,6.184,149.075
C09919=1156.541,33.861,-49.146,-179.857,6.185,149.074
C09920=1156.536,34.110,-49.161,-179.855,6.186,149.074
C09921=1156.531,34.360,-49.175,-179.852,6.187,149.073
C09922=1156.526,34.610,-49.191,-179.850,6.188,149.072
C09923=1156.521,34.859,-49.205,-179.846,6.189,149.072
C09924=1156.516,35.109,-49.221,-179.844,6.190,149.071
C09925=1156.511,35.358,-49.236,-179.842,6.191,149.071
C09926=1156.506,35.607,-49.250,-179.839,6.192,149.070
C09927=1156.501,35.857,-49.266,-179.837,6.193,149.070
C09928=1156.496,36.107,-49.280,-179.834,6.193,149.069
C09929=1156.490,36.356,-49.295,-179.831,6.195,149.069
C09930=1156.486,36.605,-49.310,-179.829,6.195,149.068
C09931=1156.480,36.855,-49.325,-179.827,6.196,149.067
C09932=1156.475,37.104,-49.340,-179.823,6.197,149.067
C09933=1156.470,37.354,-49.356,-179.821,6.198,149.066
C09934=1156.466,37.604,-49.371,-179.819,6.199,149.066
C09935=1156.461,37.853,-49.386,-179.816,6.200,149.065
C09936=1156.456,38.102,-49.401,-179.813,6.201,149.065
C09937=1156.451,38.352,-49.415,-179.811,6.202,149.064
C09938=1156.445,38.602,-49.431,-179.808,6.203,149.063
C09939=1156.441,38.851,-49.446,-179.806,6.204,149.063
C09940=1156.435,39.100,-49.462,-179.803,6.204,149.062
C09941=1156.430,39.350,-49.476,-179.800,6.206,149.062
C09942=1156.425,39.599,-49.491,-179.798,6.207,149.061
C09943=1156.420,39.848,-49.506,-179.795,6.207,149.061
C09944=1156.415,40.098,-49.522,-179.793,6.209,149.060
C09945=1156.410,40.348,-49.537,-179.790,6.209,149.060
C09946=1156.405,40.598,-49.552,-179.787,6.211,149.059
C09947=1156.400,40.847,-49.568,-179.785,6.211,149.058
C09948=1156.395,41.096,-49.583,-179.782,6.212,149.058
C09949=1156.390,41.345,-49.598,-179.779,6.214,149.057
C09950=1156.385,41.595,-49.613,-179.777,6.214,149.057
C09951=1156.380,41.845,-49.629,-179.774,6.215,149.056
C09952=1156.375,42.094,-49.644,-179.772,6.217,149.056
C09953=1156.370,42.344,-49.659,-179.769,6.217,149.055
C09954=1156.364,42.593,-49.675,-179.766,6.219,149.055
C09955=1156.360,42.842,-49.690,-179.764,6.220,149.054
C09956=1156.354,43.092,-49.705,-179.761,6.220,149.054
C09957=1156.350,43.342,-49.720,-179.759,6.222,149.053
C09958=1156.345,43.591,-49.736,-179.756,6.222,149.052
C09959=1156.339,43.841,-49.751,-179.754,6.223,149.052
C09960=1156.335,44.090,-49.766,-179.751,6.224,149.051
C09961=1156.329,44.339,-49.782,-179.748,6.225,149.051
C09962=1156.324,44.589,-49.798,-179.745,6.226,149.050
C09963=1156.320,44.839,-49.813,-179.743,6.227,149.050
C09964=1156.314,45.088,-49.828,-179.740,6.228,149.049
C09965=1156.310,45.337,-49.843,-179.738,6.229,149.049
C09966=1156.305,45.587,-49.859,-179.736,6.230,149.048
C09967=1156.300,45.837,-49.875,-179.732,6.232,149.048
C09968=1156.294,46.086,-49.890,-179.730,6.232,149.047
C09969=1156.290,46.335,-49.905,-179.728,6.233,149.046
C09970=1156.284,46.584,-49.921,-179.725,6.235,149.046
C09971=1156.279,46.835,-49.937,-179.722,6.235,149.045
C09972=1156.275,47.084,-49.952,-179.719,6.237,149.045
C09973=1156.269,47.333,-49.968,-179.717,6.237,149.044
C09974=1156.264,47.582,-49.983,-179.715,6.238,149.044
C09975=1156.260,47.832,-49.999,-179.712,6.240,149.043
C09976=1156.255,48.082,-50.014,-179.709,6.240,149.043
C09977=1156.249,48.331,-50.030,-179.706,6.242,149.042
C09978=1156.244,48.581,-50.046,-179.704,6.242,149.042
C09979=1156.240,48.830,-50.061,-179.702,6.243,149.041
C09980=1156.235,49.079,-50.077,-179.698,6.244,149.040
C09981=1156.229,49.328,-50.093,-179.696,6.245,149.040
C09982=1156.224,49.578,-50.108,-179.693,6.247,149.039
C09983=1156.220,49.828,-50.123,-179.691,6.247,149.039
C09984=1156.214,50.077,-50.139,-179.688,6.249,149.038
C09985=1156.210,50.327,-50.155,-179.685,6.250,149.038
C09986=1156.204,50.576,-50.171,-179.683,6.250,149.037
C09987=1156.199,50.825,-50.187,-179.680,6.252,149.037
C09988=1156.195,51.075,-50.202,-179.678,6.253,149.036
C09989=1156.190,51.324,-50.218,-179.675,6.254,149.036
C09990=1156.184,51.574,-50.233,-179.673,6.255,149.035
C09991=1156.180,51.824,-50.249,-179.669,6.256,149.034
C09992=1156.174,52.073,-50.266,-179.667,6.257,149.034
C09993=1156.170,52.322,-50.281,-179.665,6.258,149.034
C09994=1156.165,52.572,-50.297,-179.662,6.259,149.033
C09995=1156.160,52.821,-50.312,-179.660,6.260,149.032
C09996=1156.155,53.070,-50.329,-179.656,6.261,149.032
//INST
///DATE 2021/06/15 17:26
///ATTR SC,RW,RJ
////FRAME ROBOT
///GROUP1 RB1
NOP
MOVL C00000 V=800.0 PL=0
MOVL C00001 V=800.0 PL=0
MOVL C00002 V=800.0 PL=0
MOVL C00003 V=800.0 PL=0
MOVL C00004 V=800.0 PL=0
MOVL C00005 V=800.0 PL=0
MOVL C00006 V=800.0 PL=0
MOVL C00007 V=800.0 PL=0
MOVL C00008 V=800.0 PL=0
MOVL C00009 V=800.0 PL=0
MOVL C00010 V=800.0 PL=0
MOVL C00011 V=800.0 PL=0
MOVL C00012 V=800.0 PL=0
MOVL C00013 V=800.0 PL=0
MOVL C00014 V=800.0 PL=0
MOVL C00015 V=800.0 PL=0
MOVL C00016 V=800.0 PL=0
MOVL C00017 V=800.0 PL=0
MOVL C00018 V=800.0 PL=0
MOVL C00019 V=800.0 PL=0
MOVL C00020 V=800.0 PL=0
MOVL C00021 V=800.0 PL=0
MOVL C00022 V=800.0 PL=0
MOVL C00023 V=800.0 PL=0
MOVL C00024 V=800.0 PL=0
MOVL C00025 V=800.0 PL=0
MOVL C00026 V=800.0 PL=0
MOVL C00027 V=800.0 PL=0
MOVL C00028 V=800.0 PL=0
MOVL C00029 V=800.0 PL=0
MOVL C00030 V=800.0 PL=0
MOVL C00031 V=800.0 PL=0
MOVL C00032 V=800.0 PL=0
MOVL C00033 V=800.0 PL=0
MOVL C00034 V=800.0 PL=0
MOVL C00035 V=800.0 PL=0
MOVL C00036 V=800.0 PL=0
MOVL C00037 V=800.0 PL=0
MOVL C00038 V=800.0 PL=0
MOVL C00039 V=800.0 PL=0
MOVL C00040 V=800.0 PL=0
MOVL C00041 V=800.0 PL=0
MOVL C00042 V=800.0 PL=0
MOVL C00043 V=800.0 PL=0
MOVL C00044 V=800.0 PL=0
MOVL C00045 V=800.0 PL=0
MOVL C00046 V=800.0 PL=0
MOVL C00047 V=800.0 PL=0
MOVL C00048 V=800.0 PL=0
MOVL C00049 V=800.0 PL=0
MOVL C00050 V=800.0 PL=0
MOVL C00051 V=800.0 PL=0
MOVL C00052 V=800.0 PL=0
MOVL C00053 V=800.0 PL=0
MOVL C00054 V=800.0 PL=0
MOVL C00055 V=800.0 PL=0
MOVL C00056 V=800.0 PL=0
MOVL C00057 V=800.0 PL=0
MOVL C00058 V=800.0 PL=0
MOVL C00059 V=800.0 PL=0
MOVL C00060 V=800.0 PL=0
MOVL C00061 V=800.0 PL=0
MOVL C00062 V=800.0 PL=0
MOVL C00063 V=800.0 PL=0
MOVL C00064 V=800.0 PL=0
MOVL C00065 V=800.0 PL=0
MOVL C00066 V=800.0 PL=0
MOVL C00067 V=800.0 PL=0
MOVL C00068 V=800.0 PL=0
MOVL C00069 V=800.0 PL=0
MOVL C00070 V=800.0 PL=0
MOVL C00071 V=800.0 PL=0
MOVL C00072 V=800.0 PL=0
MOVL C00073 V=800.0 PL=0
MOVL C00074 V=800.0 PL=0
MOVL C00075 V=800.0 PL=0
MOVL C00076 V=800.0 PL=0
MOVL C00077 V=800.0 PL=0
MOVL C00078 V=800.0 PL=0
MOVL C00079 V=800.0 PL=0
MOVL C00080 V=800.0 PL=0
MOVL C00081 V=800.0 PL=0
MOVL C00082 V=800.0 PL=0
MOVL C00083 V=800.0 PL=0
MOVL C00084 V=800.0 PL=0
MOVL C00085 V=800.0 PL=0
MOVL C00086 V=800.0 PL=0
MOVL C00087 V=800.0 PL=0
MOVL C00088 V=800.0 PL=0
MOVL C00089 V=800.0 PL=0
MOVL C00090 V=800.0 PL=0
MOVL C00091 V=800.0 PL=0
MOVL C00092 V=800.0 PL=0
MOVL C00093 V=800.0 PL=0
MOVL C00094 V=800.0 PL=0
MOVL C00095 V=800.0 PL=0
MOVL C00096 V=800.0 PL=0
MOVL C00097 V=800.0 PL=0
MOVL C00098 V=800.0 PL=0
MOVL C00099 V=800.0 PL=0
MOVL C00100 V=800.0 PL=0
MOVL C00101 V=800.0 PL=0
MOVL C00102 V=800.0 PL=0
MOVL C00103 V=800.0 PL=0
MOVL C00104 V=800.0 PL=0
MOVL C00105 V=800.0 PL=0
MOVL C00106 V=800.0 PL=0
MOVL C00107 V=800.0 PL=0
MOVL C00108 V=800.0 PL=0
MOVL C00109 V=800.0 PL=0
MOVL C00110 V=800.0 PL=0
MOVL C00111 V=800.0 PL=0
MOVL C00112 V=800.0 PL=0
MOVL C00113 V=800.0 PL=0
MOVL C00114 V=800.0 PL=0
MOVL C00115 V=800.0 PL=0
MOVL C00116 V=800.0 PL=0
MOVL C00117 V=800.0 PL=0
MOVL C00118 V=800.0 PL=0
MOVL C00119 V=800.0 PL=0
MOVL C00120 V=800.0 PL=0
MOVL C00121 V=800.0 PL=0
MOVL C00122 V=800.0 PL=0
MOVL C00123 V=800.0 PL=0
MOVL C00124 V=800.0 PL=0
MOVL C00125 V=800.0 PL=0
MOVL C00126 V=800.0 PL=0
MOVL C00127 V=800.0 PL=0
MOVL C00128 V=800.0 PL=0
MOVL C00129 V=800.0 PL=0
MOVL C00130 V=800.0 PL=0
MOVL C00131 V=800.0 PL=0
MOVL C00132 V=800.0 PL=0
MOVL C00133 V=800.0 PL=0
MOVL C00134 V=800.0 PL=0
MOVL C00135 V=800.0 PL=0
MOVL C00136 V=800.0 PL=0
MOVL C00137 V=800.0 PL=0
MOVL C00138 V=800.0 PL=0
MOVL C00139 V=800.0 PL=0
MOVL C00140 V=800.0 PL=0
MOVL C00141 V=800.0 PL=0
MOVL C00142 V=800.0 PL=0
MOVL C00143 V=800.0 PL=0
MOVL C00144 V=800.0 PL=0
MOVL C00145 V=800.0 PL=0
MOVL C00146 V=800.0 PL=0
MOVL C00147 V=800.0 PL=0
MOVL C00148 V=800.0 PL=0
MOVL C00149 V=800.0 PL=0
MOVL C00150 V=800.0 PL=0
MOVL C00151 V=800.0 PL=0
MOVL C00152 V=800.0 PL=0
MOVL C00153 V=800.0 PL=0
MOVL C00154 V=800.0 PL=0
MOVL C00155 V=800.0 PL=0
MOVL C00156 V=800.0 PL=0
MOVL C00157 V=800.0 PL=0
MOVL C00158 V=800.0 PL=0
MOVL C00159 V=800.0 PL=0
MOVL C00160 V=800.0 PL=0
MOVL C00161 V=800.0 PL=0
MOVL C00162 V=800.0 PL=0
MOVL C00163 V=800.0 PL=0
MOVL C00164 V=800.0 PL=0
MOVL C00165 V=800.0 PL=0
MOVL C00166 V=800.0 PL=0
MOVL C00167 V=800.0 PL=0
MOVL C00168 V=800.0 PL=0
MOVL C00169 V=800.0 PL=0
MOVL C00170 V=800.0 PL=0
MOVL C00171 V=800.0 PL=0
MOVL C00172 V=800.0 PL=0
MOVL C00173 V=800.0 PL=0
MOVL C00174 V=800.0 PL=0
MOVL C00175 V=800.0 PL=0
MOVL C00176 V=800.0 PL=0
MOVL C00177 V=800.0 PL=0
MOVL C00178 V=800.0 PL=0
MOVL C00179 V=800.0 PL=0
MOVL C00180 V=800.0 PL=0
MOVL C00181 V=800.0 PL=0
MOVL C00182 V=800.0 PL=0
MOVL C00183 V=800.0 PL=0
MOVL C00184 V=800.0 PL=0
MOVL C00185 V=800.0 PL=0
MOVL C00186 V=800.0 PL=0
MOVL C00187 V=800.0 PL=0
MOVL C00188 V=800.0 PL=0
MOVL C00189 V=800.0 PL=0
MOVL C00190 V=800.0 PL=0
MOVL C00191 V=800.0 PL=0
MOVL C00192 V=800.0 PL=0
MOVL C00193 V=800.0 PL=0
MOVL C00194 V=800.0 PL=0
MOVL C00195 V=800.0 PL=0
MOVL C00196 V=800.0 PL=0
MOVL C00197 V=800.0 PL=0
MOVL C00198 V=800.0 PL=0
MOVL C00199 V=800.0 PL=0
MOVL C00200 V=800.0 PL=0
MOVL C00201 V=800.0 PL=0
MOVL C00202 V=800.0 PL=0
MOVL C00203 V=800.0 PL=0
MOVL C00204 V=800.0 PL=0
MOVL C00205 V=800.0 PL=0
MOVL C00206 V=800.0 PL=0
MOVL C00207 V=800.0 PL=0
MOVL C00208 V=800.0 PL=0
MOVL C00209 V=800.0 PL=0
MOVL C00210 V=800.0 PL=0
MOVL C00211 V=800.0 PL=0
MOVL C00212 V=800.0 PL=0
MOVL C00213 V=800.0 PL=0
MOVL C00214 V=800.0 PL=0
MOVL C00215 V=800.0 PL=0
MOVL C00216 V=800.0 PL=0
MOVL C00217 V=800.0 PL=0
MOVL C00218 V=800.0 PL=0
MOVL C00219 V=800.0 PL=0
MOVL C00220 V=800.0 PL=0
MOVL C00221 V=800.0 PL=0
MOVL C00222 V=800.0 PL=0
MOVL C00223 V=800.0 PL=0
MOVL C00224 V=800.0 PL=0
MOVL C00225 V=800.0 PL=0
MOVL C00226 V=800.0 PL=0
MOVL C00227 V=800.0 PL=0
MOVL C00228 V=800.0 PL=0
MOVL C00229 V=800.0 PL=0
MOVL C00230 V=800.0 PL=0
MOVL C00231 V=800.0 PL=0
MOVL C00232 V=800.0 PL=0
MOVL C00233 V=800.0 PL=0
MOVL C00234 V=800.0 PL=0
MOVL C00235 V=800.0 PL=0
MOVL C00236 V=800.0 PL=0
MOVL C00237 V=800.0 PL=0
MOVL C00238 V=800.0 PL=0
MOVL C00239 V=800.0 PL=0
MOVL C00240 V=800.0 PL=0
MOVL C00241 V=800.0 PL=0
MOVL C00242 V=800.0 PL=0
MOVL C00243 V=800.0 PL=0
MOVL C00244 V=800.0 PL=0
MOVL C00245 V=800.0 PL=0
MOVL C00246 V=800.0 PL=0
MOVL C00247 V=800.0 PL=0
MOVL C00248 V=800.0 PL=0
MOVL C00249 V=800.0 PL=0
MOVL C00250 V=800.0 PL=0
MOVL C00251 V=800.0 PL=0
MOVL C00252 V=800.0 PL=0
MOVL C00253 V=800.0 PL=0
MOVL C00254 V=800.0 PL=0
MOVL C00255 V=800.0 PL=0
MOVL C00256 V=800.0 PL=0
MOVL C00257 V=800.0 PL=0
MOVL C00258 V=800.0 PL=0
MOVL C00259 V=800.0 PL=0
MOVL C00260 V=800.0 PL=0
MOVL C00261 V=800.0 PL=0
MOVL C00262 V=800.0 PL=0
MOVL C00263 V=800.0 PL=0
MOVL C00264 V=800.0 PL=0
MOVL C00265 V=800.0 PL=0
MOVL C00266 V=800.0 PL=0
MOVL C00267 V=800.0 PL=0
MOVL C00268 V=800.0 PL=0
MOVL C00269 V=800.0 PL=0
MOVL C00270 V=800.0 PL=0
MOVL C00271 V=800.0 PL=0
MOVL C00272 V=800.0 PL=0
MOVL C00273 V=800.0 PL=0
MOVL C00274 V=800.0 PL=0
MOVL C00275 V=800.0 PL=0
MOVL C00276 V=800.0 PL=0
MOVL C00277 V=800.0 PL=0
MOVL C00278 V=800.0 PL=0
MOVL C00279 V=800.0 PL=0
MOVL C00280 V=800.0 PL=0
MOVL C00281 V=800.0 PL=0
MOVL C00282 V=800.0 PL=0
MOVL C00283 V=800.0 PL=0
MOVL C00284 V=800.0 PL=0
MOVL C00285 V=800.0 PL=0
MOVL C00286 V=800.0 PL=0
MOVL C00287 V=800.0 PL=0
MOVL C00288 V=800.0 PL=0
MOVL C00289 V=800.0 PL=0
MOVL C00290 V=800.0 PL=0
MOVL C00291 V=800.0 PL=0
MOVL C00292 V=800.0 PL=0
MOVL C00293 V=800.0 PL=0
MOVL C00294 V=800.0 PL=0
MOVL C00295 V=800.0 PL=0
MOVL C00296 V=800.0 PL=0
MOVL C00297 V=800.0 PL=0
MOVL C00298 V=800.0 PL=0
MOVL C00299 V=800.0 PL=0
MOVL C00300 V=800.0 PL=0
MOVL C00301 V=800.0 PL=0
MOVL C00302 V=800.0 PL=0
MOVL C00303 V=800.0 PL=0
MOVL C00304 V=800.0 PL=0
MOVL C00305 V=800.0 PL=0
MOVL C00306 V=800.0 PL=0
MOVL C00307 V=800.0 PL=0
MOVL C00308 V=800.0 PL=0
MOVL C00309 V=800.0 PL=0
MOVL C00310 V=800.0 PL=0
MOVL C00311 V=800.0 PL=0
MOVL C00312 V=800.0 PL=0
MOVL C00313 V=800.0 PL=0
MOVL C00314 V=800.0 PL=0
MOVL C00315 V=800.0 PL=0
MOVL C00316 V=800.0 PL=0
MOVL C00317 V=800.0 PL=0
MOVL C00318 V=800.0 PL=0
MOVL C00319 V=800.0 PL=0
MOVL C00320 V=800.0 PL=0
MOVL C00321 V=800.0 PL=0
MOVL C00322 V=800.0 PL=0
MOVL C00323 V=800.0 PL=0
MOVL C00324 V=800.0 PL=0
MOVL C00325 V=800.0 PL=0
MOVL C00326 V=800.0 PL=0
MOVL C00327 V=800.0 PL=0
MOVL C00328 V=800.0 PL=0
MOVL C00329 V=800.0 PL=0
MOVL C00330 V=800.0 PL=0
MOVL C00331 V=800.0 PL=0
MOVL C00332 V=800.0 PL=0
MOVL C00333 V=800.0 PL=0
MOVL C00334 V=800.0 PL=0
MOVL C00335 V=800.0 PL=0
MOVL C00336 V=800.0 PL=0
MOVL C00337 V=800.0 PL=0
MOVL C00338 V=800.0 PL=0
MOVL C00339 V=800.0 PL=0
MOVL C00340 V=800.0 PL=0
MOVL C00341 V=800.0 PL=0
MOVL C00342 V=800.0 PL=0
MOVL C00343 V=800.0 PL=0
MOVL C00344 V=800.0 PL=0
MOVL C00345 V=800.0 PL=0
MOVL C00346 V=800.0 PL=0
MOVL C00347 V=800.0 PL=0
MOVL C00348 V=800.0 PL=0
MOVL C00349 V=800.0 PL=0
MOVL C00350 V=800.0 PL=0
MOVL C00351 V=800.0 PL=0
MOVL C00352 V=800.0 PL=0
MOVL C00353 V=800.0 PL=0
MOVL C00354 V=800.0 PL=0
MOVL C00355 V=800.0 PL=0
MOVL C00356 V=800.0 PL=0
MOVL C00357 V=800.0 PL=0
MOVL C00358 V=800.0 PL=0
MOVL C00359 V=800.0 PL=0
MOVL C00360 V=800.0 PL=0
MOVL C00361 V=800.0 PL=0
MOVL C00362 V=800.0 PL=0
MOVL C00363 V=800.0 PL=0
MOVL C00364 V=800.0 PL=0
MOVL C00365 V=800.0 PL=0
MOVL C00366 V=800.0 PL=0
MOVL C00367 V=800.0 PL=0
MOVL C00368 V=800.0 PL=0
MOVL C00369 V=800.0 PL=0
MOVL C00370 V=800.0 PL=0
MOVL C00371 V=800.0 PL=0
MOVL C00372 V=800.0 PL=0
MOVL C00373 V=800.0 PL=0
MOVL C00374 V=800.0 PL=0
MOVL C00375 V=800.0 PL=0
MOVL C00376 V=800.0 PL=0
MOVL C00377 V=800.0 PL=0
MOVL C00378 V=800.0 PL=0
MOVL C00379 V=800.0 PL=0
MOVL C00380 V=800.0 PL=0
MOVL C00381 V=800.0 PL=0
MOVL C00382 V=800.0 PL=0
MOVL C00383 V=800.0 PL=0
MOVL C00384 V=800.0 PL=0
MOVL C00385 V=800.0 PL=0
MOVL C00386 V=800.0 PL=0
MOVL C00387 V=800.0 PL=0
MOVL C00388 V=800.0 PL=0
MOVL C00389 V=800.0 PL=0
MOVL C00390 V=800.0 PL=0
MOVL C00391 V=800.0 PL=0
MOVL C00392 V=800.0 PL=0
MOVL C00393 V=800.0 PL=0
MOVL C00394 V=800.0 PL=0
MOVL C00395 V=800.0 PL=0
MOVL C00396 V=800.0 PL=0
MOVL C00397 V=800.0 PL=0
MOVL C00398 V=800.0 PL=0
MOVL C00399 V=800.0 PL=0
MOVL C00400 V=800.0 PL=0
MOVL C00401 V=800.0 PL=0
MOVL C00402 V=800.0 PL=0
MOVL C00403 V=800.0 PL=0
MOVL C00404 V=800.0 PL=0
MOVL C00405 V=800.0 PL=0
MOVL C00406 V=800.0 PL=0
MOVL C00407 V=800.0 PL=0
MOVL C00408 V=800.0 PL=0
MOVL C00409 V=800.0 PL=0
MOVL C00410 V=800.0 PL=0
MOVL C00411 V=800.0 PL=0
MOVL C00412 V=800.0 PL=0
MOVL C00413 V=800.0 PL=0
MOVL C00414 V=800.0 PL=0
MOVL C00415 V=800.0 PL=0
MOVL C00416 V=800.0 PL=0
MOVL C00417 V=800.0 PL=0
MOVL C00418 V=800.0 PL=0
MOVL C00419 V=800.0 PL=0
MOVL C00420 V=800.0 PL=0
MOVL C00421 V=800.0 PL=0
MOVL C00422 V=800.0 PL=0
MOVL C00423 V=800.0 PL=0
MOVL C00424 V=800.0 PL=0
MOVL C00425 V=800.0 PL=0
MOVL C00426 V=800.0 PL=0
MOVL C00427 V=800.0 PL=0
MOVL C00428 V=800.0 PL=0
MOVL C00429 V=800.0 PL=0
MOVL C00430 V=800.0 PL=0
MOVL C00431 V=800.0 PL=0
MOVL C00432 V=800.0 PL=0
MOVL C00433 V=800.0 PL=0
MOVL C00434 V=800.0 PL=0
MOVL C00435 V=800.0 PL=0
MOVL C00436 V=800.0 PL=0
MOVL C00437 V=800.0 PL=0
MOVL C00438 V=800.0 PL=0
MOVL C00439 V=800.0 PL=0
MOVL C00440 V=800.0 PL=0
MOVL C00441 V=800.0 PL=0
MOVL C00442 V=800.0 PL=0
MOVL C00443 V=800.0 PL=0
MOVL C00444 V=800.0 PL=0
MOVL C00445 V=800.0 PL=0
MOVL C00446 V=800.0 PL=0
MOVL C00447 V=800.0 PL=0
MOVL C00448 V=800.0 PL=0
MOVL C00449 V=800.0 PL=0
MOVL C00450 V=800.0 PL=0
MOVL C00451 V=800.0 PL=0
MOVL C00452 V=800.0 PL=0
MOVL C00453 V=800.0 PL=0
MOVL C00454 V=800.0 PL=0
MOVL C00455 V=800.0 PL=0
MOVL C00456 V=800.0 PL=0
MOVL C00457 V=800.0 PL=0
MOVL C00458 V=800.0 PL=0
MOVL C00459 V=800.0 PL=0
MOVL C00460 V=800.0 PL=0
MOVL C00461 V=800.0 PL=0
MOVL C00462 V=800.0 PL=0
MOVL C00463 V=800.0 PL=0
MOVL C00464 V=800.0 PL=0
MOVL C00465 V=800.0 PL=0
MOVL C00466 V=800.0 PL=0
MOVL C00467 V=800.0 PL=0
MOVL C00468 V=800.0 PL=0
MOVL C00469 V=800.0 PL=0
MOVL C00470 V=800.0 PL=0
MOVL C00471 V=800.0 PL=0
MOVL C00472 V=800.0 PL=0
MOVL C00473 V=800.0 PL=0
MOVL C00474 V=800.0 PL=0
MOVL C00475 V=800.0 PL=0
MOVL C00476 V=800.0 PL=0
MOVL C00477 V=800.0 PL=0
MOVL C00478 V=800.0 PL=0
MOVL C00479 V=800.0 PL=0
MOVL C00480 V=800.0 PL=0
MOVL C00481 V=800.0 PL=0
MOVL C00482 V=800.0 PL=0
MOVL C00483 V=800.0 PL=0
MOVL C00484 V=800.0 PL=0
MOVL C00485 V=800.0 PL=0
MOVL C00486 V=800.0 PL=0
MOVL C00487 V=800.0 PL=0
MOVL C00488 V=800.0 PL=0
MOVL C00489 V=800.0 PL=0
MOVL C00490 V=800.0 PL=0
MOVL C00491 V=800.0 PL=0
MOVL C00492 V=800.0 PL=0
MOVL C00493 V=800.0 PL=0
MOVL C00494 V=800.0 PL=0
MOVL C00495 V=800.0 PL=0
MOVL C00496 V=800.0 PL=0
MOVL C00497 V=800.0 PL=0
MOVL C00498 V=800.0 PL=0
MOVL C00499 V=800.0 PL=0
MOVL C00500 V=800.0 PL=0
MOVL C00501 V=800.0 PL=0
MOVL C00502 V=800.0 PL=0
MOVL C00503 V=800.0 PL=0
MOVL C00504 V=800.0 PL=0
MOVL C00505 V=800.0 PL=0
MOVL C00506 V=800.0 PL=0
MOVL C00507 V=800.0 PL=0
MOVL C00508 V=800.0 PL=0
MOVL C00509 V=800.0 PL=0
MOVL C00510 V=800.0 PL=0
MOVL C00511 V=800.0 PL=0
MOVL C00512 V=800.0 PL=0
MOVL C00513 V=800.0 PL=0
MOVL C00514 V=800.0 PL=0
MOVL C00515 V=800.0 PL=0
MOVL C00516 V=800.0 PL=0
MOVL C00517 V=800.0 PL=0
MOVL C00518 V=800.0 PL=0
MOVL C00519 V=800.0 PL=0
MOVL C00520 V=800.0 PL=0
MOVL C00521 V=800.0 PL=0
MOVL C00522 V=800.0 PL=0
MOVL C00523 V=800.0 PL=0
MOVL C00524 V=800.0 PL=0
MOVL C00525 V=800.0 PL=0
MOVL C00526 V=800.0 PL=0
MOVL C00527 V=800.0 PL=0
MOVL C00528 V=800.0 PL=0
MOVL C00529 V=800.0 PL=0
MOVL C00530 V=800.0 PL=0
MOVL C00531 V=800.0 PL=0
MOVL C00532 V=800.0 PL=0
MOVL C00533 V=800.0 PL=0
MOVL C00534 V=800.0 PL=0
MOVL C00535 V=800.0 PL=0
MOVL C00536 V=800.0 PL=0
MOVL C00537 V=800.0 PL=0
MOVL C00538 V=800.0 PL=0
MOVL C00539 V=800.0 PL=0
MOVL C00540 V=800.0 PL=0
MOVL C00541 V=800.0 PL=0
MOVL C00542 V=800.0 PL=0
MOVL C00543 V=800.0 PL=0
MOVL C00544 V=800.0 PL=0
MOVL C00545 V=800.0 PL=0
MOVL C00546 V=800.0 PL=0
MOVL C00547 V=800.0 PL=0
MOVL C00548 V=800.0 PL=0
MOVL C00549 V=800.0 PL=0
MOVL C00550 V=800.0 PL=0
MOVL C00551 V=800.0 PL=0
MOVL C00552 V=800.0 PL=0
MOVL C00553 V=800.0 PL=0
MOVL C00554 V=800.0 PL=0
MOVL C00555 V=800.0 PL=0
MOVL C00556 V=800.0 PL=0
MOVL C00557 V=800.0 PL=0
MOVL C00558 V=800.0 PL=0
MOVL C00559 V=800.0 PL=0
MOVL C00560 V=800.0 PL=0
MOVL C00561 V=800.0 PL=0
MOVL C00562 V=800.0 PL=0
MOVL C00563 V=800.0 PL=0
MOVL C00564 V=800.0 PL=0
MOVL C00565 V=800.0 PL=0
MOVL C00566 V=800.0 PL=0
MOVL C00567 V=800.0 PL=0
MOVL C00568 V=800.0 PL=0
MOVL C00569 V=800.0 PL=0
MOVL C00570 V=800.0 PL=0
MOVL C00571 V=800.0 PL=0
MOVL C00572 V=800.0 PL=0
MOVL C00573 V=800.0 PL=0
MOVL C00574 V=800.0 PL=0
MOVL C00575 V=800.0 PL=0
MOVL C00576 V=800.0 PL=0
MOVL C00577 V=800.0 PL=0
MOVL C00578 V=800.0 PL=0
MOVL C00579 V=800.0 PL=0
MOVL C00580 V=800.0 PL=0
MOVL C00581 V=800.0 PL=0
MOVL C00582 V=800.0 PL=0
MOVL C00583 V=800.0 PL=0
MOVL C00584 V=800.0 PL=0
MOVL C00585 V=800.0 PL=0
MOVL C00586 V=800.0 PL=0
MOVL C00587 V=800.0 PL=0
MOVL C00588 V=800.0 PL=0
MOVL C00589 V=800.0 PL=0
MOVL C00590 V=800.0 PL=0
MOVL C00591 V=800.0 PL=0
MOVL C00592 V=800.0 PL=0
MOVL C00593 V=800.0 PL=0
MOVL C00594 V=800.0 PL=0
MOVL C00595 V=800.0 PL=0
MOVL C00596 V=800.0 PL=0
MOVL C00597 V=800.0 PL=0
MOVL C00598 V=800.0 PL=0
MOVL C00599 V=800.0 PL=0
MOVL C00600 V=800.0 PL=0
MOVL C00601 V=800.0 PL=0
MOVL C00602 V=800.0 PL=0
MOVL C00603 V=800.0 PL=0
MOVL C00604 V=800.0 PL=0
MOVL C00605 V=800.0 PL=0
MOVL C00606 V=800.0 PL=0
MOVL C00607 V=800.0 PL=0
MOVL C00608 V=800.0 PL=0
MOVL C00609 V=800.0 PL=0
MOVL C00610 V=800.0 PL=0
MOVL C00611 V=800.0 PL=0
MOVL C00612 V=800.0 PL=0
MOVL C00613 V=800.0 PL=0
MOVL C00614 V=800.0 PL=0
MOVL C00615 V=800.0 PL=0
MOVL C00616 V=800.0 PL=0
MOVL C00617 V=800.0 PL=0
MOVL C00618 V=800.0 PL=0
MOVL C00619 V=800.0 PL=0
MOVL C00620 V=800.0 PL=0
MOVL C00621 V=800.0 PL=0
MOVL C00622 V=800.0 PL=0
MOVL C00623 V=800.0 PL=0
MOVL C00624 V=800.0 PL=0
MOVL C00625 V=800.0 PL=0
MOVL C00626 V=800.0 PL=0
MOVL C00627 V=800.0 PL=0
MOVL C00628 V=800.0 PL=0
MOVL C00629 V=800.0 PL=0
MOVL C00630 V=800.0 PL=0
MOVL C00631 V=800.0 PL=0
MOVL C00632 V=800.0 PL=0
MOVL C00633 V=800.0 PL=0
MOVL C00634 V=800.0 PL=0
MOVL C00635 V=800.0 PL=0
MOVL C00636 V=800.0 PL=0
MOVL C00637 V=800.0 PL=0
MOVL C00638 V=800.0 PL=0
MOVL C00639 V=800.0 PL=0
MOVL C00640 V=800.0 PL=0
MOVL C00641 V=800.0 PL=0
MOVL C00642 V=800.0 PL=0
MOVL C00643 V=800.0 PL=0
MOVL C00644 V=800.0 PL=0
MOVL C00645 V=800.0 PL=0
MOVL C00646 V=800.0 PL=0
MOVL C00647 V=800.0 PL=0
MOVL C00648 V=800.0 PL=0
MOVL C00649 V=800.0 PL=0
MOVL C00650 V=800.0 PL=0
MOVL C00651 V=800.0 PL=0
MOVL C00652 V=800.0 PL=0
MOVL C00653 V=800.0 PL=0
MOVL C00654 V=800.0 PL=0
MOVL C00655 V=800.0 PL=0
MOVL C00656 V=800.0 PL=0
MOVL C00657 V=800.0 PL=0
MOVL C00658 V=800.0 PL=0
MOVL C00659 V=800.0 PL=0
MOVL C00660 V=800.0 PL=0
MOVL C00661 V=800.0 PL=0
MOVL C00662 V=800.0 PL=0
MOVL C00663 V=800.0 PL=0
MOVL C00664 V=800.0 PL=0
MOVL C00665 V=800.0 PL=0
MOVL C00666 V=800.0 PL=0
MOVL C00667 V=800.0 PL=0
MOVL C00668 V=800.0 PL=0
MOVL C00669 V=800.0 PL=0
MOVL C00670 V=800.0 PL=0
MOVL C00671 V=800.0 PL=0
MOVL C00672 V=800.0 PL=0
MOVL C00673 V=800.0 PL=0
MOVL C00674 V=800.0 PL=0
MOVL C00675 V=800.0 PL=0
MOVL C00676 V=800.0 PL=0
MOVL C00677 V=800.0 PL=0
MOVL C00678 V=800.0 PL=0
MOVL C00679 V=800.0 PL=0
MOVL C00680 V=800.0 PL=0
MOVL C00681 V=800.0 PL=0
MOVL C00682 V=800.0 PL=0
MOVL C00683 V=800.0 PL=0
MOVL C00684 V=800.0 PL=0
MOVL C00685 V=800.0 PL=0
MOVL C00686 V=800.0 PL=0
MOVL C00687 V=800.0 PL=0
MOVL C00688 V=800.0 PL=0
MOVL C00689 V=800.0 PL=0
MOVL C00690 V=800.0 PL=0
MOVL C00691 V=800.0 PL=0
MOVL C00692 V=800.0 PL=0
MOVL C00693 V=800.0 PL=0
MOVL C00694 V=800.0 PL=0
MOVL C00695 V=800.0 PL=0
MOVL C00696 V=800.0 PL=0
MOVL C00697 V=800.0 PL=0
MOVL C00698 V=800.0 PL=0
MOVL C00699 V=800.0 PL=0
MOVL C00700 V=800.0 PL=0
MOVL C00701 V=800.0 PL=0
MOVL C00702 V=800.0 PL=0
MOVL C00703 V=800.0 PL=0
MOVL C00704 V=800.0 PL=0
MOVL C00705 V=800.0 PL=0
MOVL C00706 V=800.0 PL=0
MOVL C00707 V=800.0 PL=0
MOVL C00708 V=800.0 PL=0
MOVL C00709 V=800.0 PL=0
MOVL C00710 V=800.0 PL=0
MOVL C00711 V=800.0 PL=0
MOVL C00712 V=800.0 PL=0
MOVL C00713 V=800.0 PL=0
MOVL C00714 V=800.0 PL=0
MOVL C00715 V=800.0 PL=0
MOVL C00716 V=800.0 PL=0
MOVL C00717 V=800.0 PL=0
MOVL C00718 V=800.0 PL=0
MOVL C00719 V=800.0 PL=0
MOVL C00720 V=800.0 PL=0
MOVL C00721 V=800.0 PL=0
MOVL C00722 V=800.0 PL=0
MOVL C00723 V=800.0 PL=0
MOVL C00724 V=800.0 PL=0
MOVL C00725 V=800.0 PL=0
MOVL C00726 V=800.0 PL=0
MOVL C00727 V=800.0 PL=0
MOVL C00728 V=800.0 PL=0
MOVL C00729 V=800.0 PL=0
MOVL C00730 V=800.0 PL=0
MOVL C00731 V=800.0 PL=0
MOVL C00732 V=800.0 PL=0
MOVL C00733 V=800.0 PL=0
MOVL C00734 V=800.0 PL=0
MOVL C00735 V=800.0 PL=0
MOVL C00736 V=800.0 PL=0
MOVL C00737 V=800.0 PL=0
MOVL C00738 V=800.0 PL=0
MOVL C00739 V=800.0 PL=0
MOVL C00740 V=800.0 PL=0
MOVL C00741 V=800.0 PL=0
MOVL C00742 V=800.0 PL=0
MOVL C00743 V=800.0 PL=0
MOVL C00744 V=800.0 PL=0
MOVL C00745 V=800.0 PL=0
MOVL C00746 V=800.0 PL=0
MOVL C00747 V=800.0 PL=0
MOVL C00748 V=800.0 PL=0
MOVL C00749 V=800.0 PL=0
MOVL C00750 V=800.0 PL=0
MOVL C00751 V=800.0 PL=0
MOVL C00752 V=800.0 PL=0
MOVL C00753 V=800.0 PL=0
MOVL C00754 V=800.0 PL=0
MOVL C00755 V=800.0 PL=0
MOVL C00756 V=800.0 PL=0
MOVL C00757 V=800.0 PL=0
MOVL C00758 V=800.0 PL=0
MOVL C00759 V=800.0 PL=0
MOVL C00760 V=800.0 PL=0
MOVL C00761 V=800.0 PL=0
MOVL C00762 V=800.0 PL=0
MOVL C00763 V=800.0 PL=0
MOVL C00764 V=800.0 PL=0
MOVL C00765 V=800.0 PL=0
MOVL C00766 V=800.0 PL=0
MOVL C00767 V=800.0 PL=0
MOVL C00768 V=800.0 PL=0
MOVL C00769 V=800.0 PL=0
MOVL C00770 V=800.0 PL=0
MOVL C00771 V=800.0 PL=0
MOVL C00772 V=800.0 PL=0
MOVL C00773 V=800.0 PL=0
MOVL C00774 V=800.0 PL=0
MOVL C00775 V=800.0 PL=0
MOVL C00776 V=800.0 PL=0
MOVL C00777 V=800.0 PL=0
MOVL C00778 V=800.0 PL=0
MOVL C00779 V=800.0 PL=0
MOVL C00780 V=800.0 PL=0
MOVL C00781 V=800.0 PL=0
MOVL C00782 V=800.0 PL=0
MOVL C00783 V=800.0 PL=0
MOVL C00784 V=800.0 PL=0
MOVL C00785 V=800.0 PL=0
MOVL C00786 V=800.0 PL=0
MOVL C00787 V=800.0 PL=0
MOVL C00788 V=800.0 PL=0
MOVL C00789 V=800.0 PL=0
MOVL C00790 V=800.0 PL=0
MOVL C00791 V=800.0 PL=0
MOVL C00792 V=800.0 PL=0
MOVL C00793 V=800.0 PL=0
MOVL C00794 V=800.0 PL=0
MOVL C00795 V=800.0 PL=0
MOVL C00796 V=800.0 PL=0
MOVL C00797 V=800.0 PL=0
MOVL C00798 V=800.0 PL=0
MOVL C00799 V=800.0 PL=0
MOVL C00800 V=800.0 PL=0
MOVL C00801 V=800.0 PL=0
MOVL C00802 V=800.0 PL=0
MOVL C00803 V=800.0 PL=0
MOVL C00804 V=800.0 PL=0
MOVL C00805 V=800.0 PL=0
MOVL C00806 V=800.0 PL=0
MOVL C00807 V=800.0 PL=0
MOVL C00808 V=800.0 PL=0
MOVL C00809 V=800.0 PL=0
MOVL C00810 V=800.0 PL=0
MOVL C00811 V=800.0 PL=0
MOVL C00812 V=800.0 PL=0
MOVL C00813 V=800.0 PL=0
MOVL C00814 V=800.0 PL=0
MOVL C00815 V=800.0 PL=0
MOVL C00816 V=800.0 PL=0
MOVL C00817 V=800.0 PL=0
MOVL C00818 V=800.0 PL=0
MOVL C00819 V=800.0 PL=0
MOVL C00820 V=800.0 PL=0
MOVL C00821 V=800.0 PL=0
MOVL C00822 V=800.0 PL=0
MOVL C00823 V=800.0 PL=0
MOVL C00824 V=800.0 PL=0
MOVL C00825 V=800.0 PL=0
MOVL C00826 V=800.0 PL=0
MOVL C00827 V=800.0 PL=0
MOVL C00828 V=800.0 PL=0
MOVL C00829 V=800.0 PL=0
MOVL C00830 V=800.0 PL=0
MOVL C00831 V=800.0 PL=0
MOVL C00832 V=800.0 PL=0
MOVL C00833 V=800.0 PL=0
MOVL C00834 V=800.0 PL=0
MOVL C00835 V=800.0 PL=0
MOVL C00836 V=800.0 PL=0
MOVL C00837 V=800.0 PL=0
MOVL C00838 V=800.0 PL=0
MOVL C00839 V=800.0 PL=0
MOVL C00840 V=800.0 PL=0
MOVL C00841 V=800.0 PL=0
MOVL C00842 V=800.0 PL=0
MOVL C00843 V=800.0 PL=0
MOVL C00844 V=800.0 PL=0
MOVL C00845 V=800.0 PL=0
MOVL C00846 V=800.0 PL=0
MOVL C00847 V=800.0 PL=0
MOVL C00848 V=800.0 PL=0
MOVL C00849 V=800.0 PL=0
MOVL C00850 V=800.0 PL=0
MOVL C00851 V=800.0 PL=0
MOVL C00852 V=800.0 PL=0
MOVL C00853 V=800.0 PL=0
MOVL C00854 V=800.0 PL=0
MOVL C00855 V=800.0 PL=0
MOVL C00856 V=800.0 PL=0
MOVL C00857 V=800.0 PL=0
MOVL C00858 V=800.0 PL=0
MOVL C00859 V=800.0 PL=0
MOVL C00860 V=800.0 PL=0
MOVL C00861 V=800.0 PL=0
MOVL C00862 V=800.0 PL=0
MOVL C00863 V=800.0 PL=0
MOVL C00864 V=800.0 PL=0
MOVL C00865 V=800.0 PL=0
MOVL C00866 V=800.0 PL=0
MOVL C00867 V=800.0 PL=0
MOVL C00868 V=800.0 PL=0
MOVL C00869 V=800.0 PL=0
MOVL C00870 V=800.0 PL=0
MOVL C00871 V=800.0 PL=0
MOVL C00872 V=800.0 PL=0
MOVL C00873 V=800.0 PL=0
MOVL C00874 V=800.0 PL=0
MOVL C00875 V=800.0 PL=0
MOVL C00876 V=800.0 PL=0
MOVL C00877 V=800.0 PL=0
MOVL C00878 V=800.0 PL=0
MOVL C00879 V=800.0 PL=0
MOVL C00880 V=800.0 PL=0
MOVL C00881 V=800.0 PL=0
MOVL C00882 V=800.0 PL=0
MOVL C00883 V=800.0 PL=0
MOVL C00884 V=800.0 PL=0
MOVL C00885 V=800.0 PL=0
MOVL C00886 V=800.0 PL=0
MOVL C00887 V=800.0 PL=0
MOVL C00888 V=800.0 PL=0
MOVL C00889 V=800.0 PL=0
MOVL C00890 V=800.0 PL=0
MOVL C00891 V=800.0 PL=0
MOVL C00892 V=800.0 PL=0
MOVL C00893 V=800.0 PL=0
MOVL C00894 V=800.0 PL=0
MOVL C00895 V=800.0 PL=0
MOVL C00896 V=800.0 PL=0
MOVL C00897 V=800.0 PL=0
MOVL C00898 V=800.0 PL=0
MOVL C00899 V=800.0 PL=0
MOVL C00900 V=800.0 PL=0
MOVL C00901 V=800.0 PL=0
MOVL C00902 V=800.0 PL=0
MOVL C00903 V=800.0 PL=0
MOVL C00904 V=800.0 PL=0
MOVL C00905 V=800.0 PL=0
MOVL C00906 V=800.0 PL=0
MOVL C00907 V=800.0 PL=0
MOVL C00908 V=800.0 PL=0
MOVL C00909 V=800.0 PL=0
MOVL C00910 V=800.0 PL=0
MOVL C00911 V=800.0 PL=0
MOVL C00912 V=800.0 PL=0
MOVL C00913 V=800.0 PL=0
MOVL C00914 V=800.0 PL=0
MOVL C00915 V=800.0 PL=0
MOVL C00916 V=800.0 PL=0
MOVL C00917 V=800.0 PL=0
MOVL C00918 V=800.0 PL=0
MOVL C00919 V=800.0 PL=0
MOVL C00920 V=800.0 PL=0
MOVL C00921 V=800.0 PL=0
MOVL C00922 V=800.0 PL=0
MOVL C00923 V=800.0 PL=0
MOVL C00924 V=800.0 PL=0
MOVL C00925 V=800.0 PL=0
MOVL C00926 V=800.0 PL=0
MOVL C00927 V=800.0 PL=0
MOVL C00928 V=800.0 PL=0
MOVL C00929 V=800.0 PL=0
MOVL C00930 V=800.0 PL=0
MOVL C00931 V=800.0 PL=0
MOVL C00932 V=800.0 PL=0
MOVL C00933 V=800.0 PL=0
MOVL C00934 V=800.0 PL=0
MOVL C00935 V=800.0 PL=0
MOVL C00936 V=800.0 PL=0
MOVL C00937 V=800.0 PL=0
MOVL C00938 V=800.0 PL=0
MOVL C00939 V=800.0 PL=0
MOVL C00940 V=800.0 PL=0
MOVL C00941 V=800.0 PL=0
MOVL C00942 V=800.0 PL=0
MOVL C00943 V=800.0 PL=0
MOVL C00944 V=800.0 PL=0
MOVL C00945 V=800.0 PL=0
MOVL C00946 V=800.0 PL=0
MOVL C00947 V=800.0 PL=0
MOVL C00948 V=800.0 PL=0
MOVL C00949 V=800.0 PL=0
MOVL C00950 V=800.0 PL=0
MOVL C00951 V=800.0 PL=0
MOVL C00952 V=800.0 PL=0
MOVL C00953 V=800.0 PL=0
MOVL C00954 V=800.0 PL=0
MOVL C00955 V=800.0 PL=0
MOVL C00956 V=800.0 PL=0
MOVL C00957 V=800.0 PL=0
MOVL C00958 V=800.0 PL=0
MOVL C00959 V=800.0 PL=0
MOVL C00960 V=800.0 PL=0
MOVL C00961 V=800.0 PL=0
MOVL C00962 V=800.0 PL=0
MOVL C00963 V=800.0 PL=0
MOVL C00964 V=800.0 PL=0
MOVL C00965 V=800.0 PL=0
MOVL C00966 V=800.0 PL=0
MOVL C00967 V=800.0 PL=0
MOVL C00968 V=800.0 PL=0
MOVL C00969 V=800.0 PL=0
MOVL C00970 V=800.0 PL=0
MOVL C00971 V=800.0 PL=0
MOVL C00972 V=800.0 PL=0
MOVL C00973 V=800.0 PL=0
MOVL C00974 V=800.0 PL=0
MOVL C00975 V=800.0 PL=0
MOVL C00976 V=800.0 PL=0
MOVL C00977 V=800.0 PL=0
MOVL C00978 V=800.0 PL=0
MOVL C00979 V=800.0 PL=0
MOVL C00980 V=800.0 PL=0
MOVL C00981 V=800.0 PL=0
MOVL C00982 V=800.0 PL=0
MOVL C00983 V=800.0 PL=0
MOVL C00984 V=800.0 PL=0
MOVL C00985 V=800.0 PL=0
MOVL C00986 V=800.0 PL=0
MOVL C00987 V=800.0 PL=0
MOVL C00988 V=800.0 PL=0
MOVL C00989 V=800.0 PL=0
MOVL C00990 V=800.0 PL=0
MOVL C00991 V=800.0 PL=0
MOVL C00992 V=800.0 PL=0
MOVL C00993 V=800.0 PL=0
MOVL C00994 V=800.0 PL=0
MOVL C00995 V=800.0 PL=0
MOVL C00996 V=800.0 PL=0
MOVL C00997 V=800.0 PL=0
MOVL C00998 V=800.0 PL=0
MOVL C00999 V=800.0 PL=0
MOVL C01000 V=800.0 PL=0
MOVL C01001 V=800.0 PL=0
MOVL C01002 V=800.0 PL=0
MOVL C01003 V=800.0 PL=0
MOVL C01004 V=800.0 PL=0
MOVL C01005 V=800.0 PL=0
MOVL C01006 V=800.0 PL=0
MOVL C01007 V=800.0 PL=0
MOVL C01008 V=800.0 PL=0
MOVL C01009 V=800.0 PL=0
MOVL C01010 V=800.0 PL=0
MOVL C01011 V=800.0 PL=0
MOVL C01012 V=800.0 PL=0
MOVL C01013 V=800.0 PL=0
MOVL C01014 V=800.0 PL=0
MOVL C01015 V=800.0 PL=0
MOVL C01016 V=800.0 PL=0
MOVL C01017 V=800.0 PL=0
MOVL C01018 V=800.0 PL=0
MOVL C01019 V=800.0 PL=0
MOVL C01020 V=800.0 PL=0
MOVL C01021 V=800.0 PL=0
MOVL C01022 V=800.0 PL=0
MOVL C01023 V=800.0 PL=0
MOVL C01024 V=800.0 PL=0
MOVL C01025 V=800.0 PL=0
MOVL C01026 V=800.0 PL=0
MOVL C01027 V=800.0 PL=0
MOVL C01028 V=800.0 PL=0
MOVL C01029 V=800.0 PL=0
MOVL C01030 V=800.0 PL=0
MOVL C01031 V=800.0 PL=0
MOVL C01032 V=800.0 PL=0
MOVL C01033 V=800.0 PL=0
MOVL C01034 V=800.0 PL=0
MOVL C01035 V=800.0 PL=0
MOVL C01036 V=800.0 PL=0
MOVL C01037 V=800.0 PL=0
MOVL C01038 V=800.0 PL=0
MOVL C01039 V=800.0 PL=0
MOVL C01040 V=800.0 PL=0
MOVL C01041 V=800.0 PL=0
MOVL C01042 V=800.0 PL=0
MOVL C01043 V=800.0 PL=0
MOVL C01044 V=800.0 PL=0
MOVL C01045 V=800.0 PL=0
MOVL C01046 V=800.0 PL=0
MOVL C01047 V=800.0 PL=0
MOVL C01048 V=800.0 PL=0
MOVL C01049 V=800.0 PL=0
MOVL C01050 V=800.0 PL=0
MOVL C01051 V=800.0 PL=0
MOVL C01052 V=800.0 PL=0
MOVL C01053 V=800.0 PL=0
MOVL C01054 V=800.0 PL=0
MOVL C01055 V=800.0 PL=0
MOVL C01056 V=800.0 PL=0
MOVL C01057 V=800.0 PL=0
MOVL C01058 V=800.0 PL=0
MOVL C01059 V=800.0 PL=0
MOVL C01060 V=800.0 PL=0
MOVL C01061 V=800.0 PL=0
MOVL C01062 V=800.0 PL=0
MOVL C01063 V=800.0 PL=0
MOVL C01064 V=800.0 PL=0
MOVL C01065 V=800.0 PL=0
MOVL C01066 V=800.0 PL=0
MOVL C01067 V=800.0 PL=0
MOVL C01068 V=800.0 PL=0
MOVL C01069 V=800.0 PL=0
MOVL C01070 V=800.0 PL=0
MOVL C01071 V=800.0 PL=0
MOVL C01072 V=800.0 PL=0
MOVL C01073 V=800.0 PL=0
MOVL C01074 V=800.0 PL=0
MOVL C01075 V=800.0 PL=0
MOVL C01076 V=800.0 PL=0
MOVL C01077 V=800.0 PL=0
MOVL C01078 V=800.0 PL=0
MOVL C01079 V=800.0 PL=0
MOVL C01080 V=800.0 PL=0
MOVL C01081 V=800.0 PL=0
MOVL C01082 V=800.0 PL=0
MOVL C01083 V=800.0 PL=0
MOVL C01084 V=800.0 PL=0
MOVL C01085 V=800.0 PL=0
MOVL C01086 V=800.0 PL=0
MOVL C01087 V=800.0 PL=0
MOVL C01088 V=800.0 PL=0
MOVL C01089 V=800.0 PL=0
MOVL C01090 V=800.0 PL=0
MOVL C01091 V=800.0 PL=0
MOVL C01092 V=800.0 PL=0
MOVL C01093 V=800.0 PL=0
MOVL C01094 V=800.0 PL=0
MOVL C01095 V=800.0 PL=0
MOVL C01096 V=800.0 PL=0
MOVL C01097 V=800.0 PL=0
MOVL C01098 V=800.0 PL=0
MOVL C01099 V=800.0 PL=0
MOVL C01100 V=800.0 PL=0
MOVL C01101 V=800.0 PL=0
MOVL C01102 V=800.0 PL=0
MOVL C01103 V=800.0 PL=0
MOVL C01104 V=800.0 PL=0
MOVL C01105 V=800.0 PL=0
MOVL C01106 V=800.0 PL=0
MOVL C01107 V=800.0 PL=0
MOVL C01108 V=800.0 PL=0
MOVL C01109 V=800.0 PL=0
MOVL C01110 V=800.0 PL=0
MOVL C01111 V=800.0 PL=0
MOVL C01112 V=800.0 PL=0
MOVL C01113 V=800.0 PL=0
MOVL C01114 V=800.0 PL=0
MOVL C01115 V=800.0 PL=0
MOVL C01116 V=800.0 PL=0
MOVL C01117 V=800.0 PL=0
MOVL C01118 V=800.0 PL=0
MOVL C01119 V=800.0 PL=0
MOVL C01120 V=800.0 PL=0
MOVL C01121 V=800.0 PL=0
MOVL C01122 V=800.0 PL=0
MOVL C01123 V=800.0 PL=0
MOVL C01124 V=800.0 PL=0
MOVL C01125 V=800.0 PL=0
MOVL C01126 V=800.0 PL=0
MOVL C01127 V=800.0 PL=0
MOVL C01128 V=800.0 PL=0
MOVL C01129 V=800.0 PL=0
MOVL C01130 V=800.0 PL=0
MOVL C01131 V=800.0 PL=0
MOVL C01132 V=800.0 PL=0
MOVL C01133 V=800.0 PL=0
MOVL C01134 V=800.0 PL=0
MOVL C01135 V=800.0 PL=0
MOVL C01136 V=800.0 PL=0
MOVL C01137 V=800.0 PL=0
MOVL C01138 V=800.0 PL=0
MOVL C01139 V=800.0 PL=0
MOVL C01140 V=800.0 PL=0
MOVL C01141 V=800.0 PL=0
MOVL C01142 V=800.0 PL=0
MOVL C01143 V=800.0 PL=0
MOVL C01144 V=800.0 PL=0
MOVL C01145 V=800.0 PL=0
MOVL C01146 V=800.0 PL=0
MOVL C01147 V=800.0 PL=0
MOVL C01148 V=800.0 PL=0
MOVL C01149 V=800.0 PL=0
MOVL C01150 V=800.0 PL=0
MOVL C01151 V=800.0 PL=0
MOVL C01152 V=800.0 PL=0
MOVL C01153 V=800.0 PL=0
MOVL C01154 V=800.0 PL=0
MOVL C01155 V=800.0 PL=0
MOVL C01156 V=800.0 PL=0
MOVL C01157 V=800.0 PL=0
MOVL C01158 V=800.0 PL=0
MOVL C01159 V=800.0 PL=0
MOVL C01160 V=800.0 PL=0
MOVL C01161 V=800.0 PL=0
MOVL C01162 V=800.0 PL=0
MOVL C01163 V=800.0 PL=0
MOVL C01164 V=800.0 PL=0
MOVL C01165 V=800.0 PL=0
MOVL C01166 V=800.0 PL=0
MOVL C01167 V=800.0 PL=0
MOVL C01168 V=800.0 PL=0
MOVL C01169 V=800.0 PL=0
MOVL C01170 V=800.0 PL=0
MOVL C01171 V=800.0 PL=0
MOVL C01172 V=800.0 PL=0
MOVL C01173 V=800.0 PL=0
MOVL C01174 V=800.0 PL=0
MOVL C01175 V=800.0 PL=0
MOVL C01176 V=800.0 PL=0
MOVL C01177 V=800.0 PL=0
MOVL C01178 V=800.0 PL=0
MOVL C01179 V=800.0 PL=0
MOVL C01180 V=800.0 PL=0
MOVL C01181 V=800.0 PL=0
MOVL C01182 V=800.0 PL=0
MOVL C01183 V=800.0 PL=0
MOVL C01184 V=800.0 PL=0
MOVL C01185 V=800.0 PL=0
MOVL C01186 V=800.0 PL=0
MOVL C01187 V=800.0 PL=0
MOVL C01188 V=800.0 PL=0
MOVL C01189 V=800.0 PL=0
MOVL C01190 V=800.0 PL=0
MOVL C01191 V=800.0 PL=0
MOVL C01192 V=800.0 PL=0
MOVL C01193 V=800.0 PL=0
MOVL C01194 V=800.0 PL=0
MOVL C01195 V=800.0 PL=0
MOVL C01196 V=800.0 PL=0
MOVL C01197 V=800.0 PL=0
MOVL C01198 V=800.0 PL=0
MOVL C01199 V=800.0 PL=0
MOVL C01200 V=800.0 PL=0
MOVL C01201 V=800.0 PL=0
MOVL C01202 V=800.0 PL=0
MOVL C01203 V=800.0 PL=0
MOVL C01204 V=800.0 PL=0
MOVL C01205 V=800.0 PL=0
MOVL C01206 V=800.0 PL=0
MOVL C01207 V=800.0 PL=0
MOVL C01208 V=800.0 PL=0
MOVL C01209 V=800.0 PL=0
MOVL C01210 V=800.0 PL=0
MOVL C01211 V=800.0 PL=0
MOVL C01212 V=800.0 PL=0
MOVL C01213 V=800.0 PL=0
MOVL C01214 V=800.0 PL=0
MOVL C01215 V=800.0 PL=0
MOVL C01216 V=800.0 PL=0
MOVL C01217 V=800.0 PL=0
MOVL C01218 V=800.0 PL=0
MOVL C01219 V=800.0 PL=0
MOVL C01220 V=800.0 PL=0
MOVL C01221 V=800.0 PL=0
MOVL C01222 V=800.0 PL=0
MOVL C01223 V=800.0 PL=0
MOVL C01224 V=800.0 PL=0
MOVL C01225 V=800.0 PL=0
MOVL C01226 V=800.0 PL=0
MOVL C01227 V=800.0 PL=0
MOVL C01228 V=800.0 PL=0
MOVL C01229 V=800.0 PL=0
MOVL C01230 V=800.0 PL=0
MOVL C01231 V=800.0 PL=0
MOVL C01232 V=800.0 PL=0
MOVL C01233 V=800.0 PL=0
MOVL C01234 V=800.0 PL=0
MOVL C01235 V=800.0 PL=0
MOVL C01236 V=800.0 PL=0
MOVL C01237 V=800.0 PL=0
MOVL C01238 V=800.0 PL=0
MOVL C01239 V=800.0 PL=0
MOVL C01240 V=800.0 PL=0
MOVL C01241 V=800.0 PL=0
MOVL C01242 V=800.0 PL=0
MOVL C01243 V=800.0 PL=0
MOVL C01244 V=800.0 PL=0
MOVL C01245 V=800.0 PL=0
MOVL C01246 V=800.0 PL=0
MOVL C01247 V=800.0 PL=0
MOVL C01248 V=800.0 PL=0
MOVL C01249 V=800.0 PL=0
MOVL C01250 V=800.0 PL=0
MOVL C01251 V=800.0 PL=0
MOVL C01252 V=800.0 PL=0
MOVL C01253 V=800.0 PL=0
MOVL C01254 V=800.0 PL=0
MOVL C01255 V=800.0 PL=0
MOVL C01256 V=800.0 PL=0
MOVL C01257 V=800.0 PL=0
MOVL C01258 V=800.0 PL=0
MOVL C01259 V=800.0 PL=0
MOVL C01260 V=800.0 PL=0
MOVL C01261 V=800.0 PL=0
MOVL C01262 V=800.0 PL=0
MOVL C01263 V=800.0 PL=0
MOVL C01264 V=800.0 PL=0
MOVL C01265 V=800.0 PL=0
MOVL C01266 V=800.0 PL=0
MOVL C01267 V=800.0 PL=0
MOVL C01268 V=800.0 PL=0
MOVL C01269 V=800.0 PL=0
MOVL C01270 V=800.0 PL=0
MOVL C01271 V=800.0 PL=0
MOVL C01272 V=800.0 PL=0
MOVL C01273 V=800.0 PL=0
MOVL C01274 V=800.0 PL=0
MOVL C01275 V=800.0 PL=0
MOVL C01276 V=800.0 PL=0
MOVL C01277 V=800.0 PL=0
MOVL C01278 V=800.0 PL=0
MOVL C01279 V=800.0 PL=0
MOVL C01280 V=800.0 PL=0
MOVL C01281 V=800.0 PL=0
MOVL C01282 V=800.0 PL=0
MOVL C01283 V=800.0 PL=0
MOVL C01284 V=800.0 PL=0
MOVL C01285 V=800.0 PL=0
MOVL C01286 V=800.0 PL=0
MOVL C01287 V=800.0 PL=0
MOVL C01288 V=800.0 PL=0
MOVL C01289 V=800.0 PL=0
MOVL C01290 V=800.0 PL=0
MOVL C01291 V=800.0 PL=0
MOVL C01292 V=800.0 PL=0
MOVL C01293 V=800.0 PL=0
MOVL C01294 V=800.0 PL=0
MOVL C01295 V=800.0 PL=0
MOVL C01296 V=800.0 PL=0
MOVL C01297 V=800.0 PL=0
MOVL C01298 V=800.0 PL=0
MOVL C01299 V=800.0 PL=0
MOVL C01300 V=800.0 PL=0
MOVL C01301 V=800.0 PL=0
MOVL C01302 V=800.0 PL=0
MOVL C01303 V=800.0 PL=0
MOVL C01304 V=800.0 PL=0
MOVL C01305 V=800.0 PL=0
MOVL C01306 V=800.0 PL=0
MOVL C01307 V=800.0 PL=0
MOVL C01308 V=800.0 PL=0
MOVL C01309 V=800.0 PL=0
MOVL C01310 V=800.0 PL=0
MOVL C01311 V=800.0 PL=0
MOVL C01312 V=800.0 PL=0
MOVL C01313 V=800.0 PL=0
MOVL C01314 V=800.0 PL=0
MOVL C01315 V=800.0 PL=0
MOVL C01316 V=800.0 PL=0
MOVL C01317 V=800.0 PL=0
MOVL C01318 V=800.0 PL=0
MOVL C01319 V=800.0 PL=0
MOVL C01320 V=800.0 PL=0
MOVL C01321 V=800.0 PL=0
MOVL C01322 V=800.0 PL=0
MOVL C01323 V=800.0 PL=0
MOVL C01324 V=800.0 PL=0
MOVL C01325 V=800.0 PL=0
MOVL C01326 V=800.0 PL=0
MOVL C01327 V=800.0 PL=0
MOVL C01328 V=800.0 PL=0
MOVL C01329 V=800.0 PL=0
MOVL C01330 V=800.0 PL=0
MOVL C01331 V=800.0 PL=0
MOVL C01332 V=800.0 PL=0
MOVL C01333 V=800.0 PL=0
MOVL C01334 V=800.0 PL=0
MOVL C01335 V=800.0 PL=0
MOVL C01336 V=800.0 PL=0
MOVL C01337 V=800.0 PL=0
MOVL C01338 V=800.0 PL=0
MOVL C01339 V=800.0 PL=0
MOVL C01340 V=800.0 PL=0
MOVL C01341 V=800.0 PL=0
MOVL C01342 V=800.0 PL=0
MOVL C01343 V=800.0 PL=0
MOVL C01344 V=800.0 PL=0
MOVL C01345 V=800.0 PL=0
MOVL C01346 V=800.0 PL=0
MOVL C01347 V=800.0 PL=0
MOVL C01348 V=800.0 PL=0
MOVL C01349 V=800.0 PL=0
MOVL C01350 V=800.0 PL=0
MOVL C01351 V=800.0 PL=0
MOVL C01352 V=800.0 PL=0
MOVL C01353 V=800.0 PL=0
MOVL C01354 V=800.0 PL=0
MOVL C01355 V=800.0 PL=0
MOVL C01356 V=800.0 PL=0
MOVL C01357 V=800.0 PL=0
MOVL C01358 V=800.0 PL=0
MOVL C01359 V=800.0 PL=0
MOVL C01360 V=800.0 PL=0
MOVL C01361 V=800.0 PL=0
MOVL C01362 V=800.0 PL=0
MOVL C01363 V=800.0 PL=0
MOVL C01364 V=800.0 PL=0
MOVL C01365 V=800.0 PL=0
MOVL C01366 V=800.0 PL=0
MOVL C01367 V=800.0 PL=0
MOVL C01368 V=800.0 PL=0
MOVL C01369 V=800.0 PL=0
MOVL C01370 V=800.0 PL=0
MOVL C01371 V=800.0 PL=0
MOVL C01372 V=800.0 PL=0
MOVL C01373 V=800.0 PL=0
MOVL C01374 V=800.0 PL=0
MOVL C01375 V=800.0 PL=0
MOVL C01376 V=800.0 PL=0
MOVL C01377 V=800.0 PL=0
MOVL C01378 V=800.0 PL=0
MOVL C01379 V=800.0 PL=0
MOVL C01380 V=800.0 PL=0
MOVL C01381 V=800.0 PL=0
MOVL C01382 V=800.0 PL=0
MOVL C01383 V=800.0 PL=0
MOVL C01384 V=800.0 PL=0
MOVL C01385 V=800.0 PL=0
MOVL C01386 V=800.0 PL=0
MOVL C01387 V=800.0 PL=0
MOVL C01388 V=800.0 PL=0
MOVL C01389 V=800.0 PL=0
MOVL C01390 V=800.0 PL=0
MOVL C01391 V=800.0 PL=0
MOVL C01392 V=800.0 PL=0
MOVL C01393 V=800.0 PL=0
MOVL C01394 V=800.0 PL=0
MOVL C01395 V=800.0 PL=0
MOVL C01396 V=800.0 PL=0
MOVL C01397 V=800.0 PL=0
MOVL C01398 V=800.0 PL=0
MOVL C01399 V=800.0 PL=0
MOVL C01400 V=800.0 PL=0
MOVL C01401 V=800.0 PL=0
MOVL C01402 V=800.0 PL=0
MOVL C01403 V=800.0 PL=0
MOVL C01404 V=800.0 PL=0
MOVL C01405 V=800.0 PL=0
MOVL C01406 V=800.0 PL=0
MOVL C01407 V=800.0 PL=0
MOVL C01408 V=800.0 PL=0
MOVL C01409 V=800.0 PL=0
MOVL C01410 V=800.0 PL=0
MOVL C01411 V=800.0 PL=0
MOVL C01412 V=800.0 PL=0
MOVL C01413 V=800.0 PL=0
MOVL C01414 V=800.0 PL=0
MOVL C01415 V=800.0 PL=0
MOVL C01416 V=800.0 PL=0
MOVL C01417 V=800.0 PL=0
MOVL C01418 V=800.0 PL=0
MOVL C01419 V=800.0 PL=0
MOVL C01420 V=800.0 PL=0
MOVL C01421 V=800.0 PL=0
MOVL C01422 V=800.0 PL=0
MOVL C01423 V=800.0 PL=0
MOVL C01424 V=800.0 PL=0
MOVL C01425 V=800.0 PL=0
MOVL C01426 V=800.0 PL=0
MOVL C01427 V=800.0 PL=0
MOVL C01428 V=800.0 PL=0
MOVL C01429 V=800.0 PL=0
MOVL C01430 V=800.0 PL=0
MOVL C01431 V=800.0 PL=0
MOVL C01432 V=800.0 PL=0
MOVL C01433 V=800.0 PL=0
MOVL C01434 V=800.0 PL=0
MOVL C01435 V=800.0 PL=0
MOVL C01436 V=800.0 PL=0
MOVL C01437 V=800.0 PL=0
MOVL C01438 V=800.0 PL=0
MOVL C01439 V=800.0 PL=0
MOVL C01440 V=800.0 PL=0
MOVL C01441 V=800.0 PL=0
MOVL C01442 V=800.0 PL=0
MOVL C01443 V=800.0 PL=0
MOVL C01444 V=800.0 PL=0
MOVL C01445 V=800.0 PL=0
MOVL C01446 V=800.0 PL=0
MOVL C01447 V=800.0 PL=0
MOVL C01448 V=800.0 PL=0
MOVL C01449 V=800.0 PL=0
MOVL C01450 V=800.0 PL=0
MOVL C01451 V=800.0 PL=0
MOVL C01452 V=800.0 PL=0
MOVL C01453 V=800.0 PL=0
MOVL C01454 V=800.0 PL=0
MOVL C01455 V=800.0 PL=0
MOVL C01456 V=800.0 PL=0
MOVL C01457 V=800.0 PL=0
MOVL C01458 V=800.0 PL=0
MOVL C01459 V=800.0 PL=0
MOVL C01460 V=800.0 PL=0
MOVL C01461 V=800.0 PL=0
MOVL C01462 V=800.0 PL=0
MOVL C01463 V=800.0 PL=0
MOVL C01464 V=800.0 PL=0
MOVL C01465 V=800.0 PL=0
MOVL C01466 V=800.0 PL=0
MOVL C01467 V=800.0 PL=0
MOVL C01468 V=800.0 PL=0
MOVL C01469 V=800.0 PL=0
MOVL C01470 V=800.0 PL=0
MOVL C01471 V=800.0 PL=0
MOVL C01472 V=800.0 PL=0
MOVL C01473 V=800.0 PL=0
MOVL C01474 V=800.0 PL=0
MOVL C01475 V=800.0 PL=0
MOVL C01476 V=800.0 PL=0
MOVL C01477 V=800.0 PL=0
MOVL C01478 V=800.0 PL=0
MOVL C01479 V=800.0 PL=0
MOVL C01480 V=800.0 PL=0
MOVL C01481 V=800.0 PL=0
MOVL C01482 V=800.0 PL=0
MOVL C01483 V=800.0 PL=0
MOVL C01484 V=800.0 PL=0
MOVL C01485 V=800.0 PL=0
MOVL C01486 V=800.0 PL=0
MOVL C01487 V=800.0 PL=0
MOVL C01488 V=800.0 PL=0
MOVL C01489 V=800.0 PL=0
MOVL C01490 V=800.0 PL=0
MOVL C01491 V=800.0 PL=0
MOVL C01492 V=800.0 PL=0
MOVL C01493 V=800.0 PL=0
MOVL C01494 V=800.0 PL=0
MOVL C01495 V=800.0 PL=0
MOVL C01496 V=800.0 PL=0
MOVL C01497 V=800.0 PL=0
MOVL C01498 V=800.0 PL=0
MOVL C01499 V=800.0 PL=0
MOVL C01500 V=800.0 PL=0
MOVL C01501 V=800.0 PL=0
MOVL C01502 V=800.0 PL=0
MOVL C01503 V=800.0 PL=0
MOVL C01504 V=800.0 PL=0
MOVL C01505 V=800.0 PL=0
MOVL C01506 V=800.0 PL=0
MOVL C01507 V=800.0 PL=0
MOVL C01508 V=800.0 PL=0
MOVL C01509 V=800.0 PL=0
MOVL C01510 V=800.0 PL=0
MOVL C01511 V=800.0 PL=0
MOVL C01512 V=800.0 PL=0
MOVL C01513 V=800.0 PL=0
MOVL C01514 V=800.0 PL=0
MOVL C01515 V=800.0 PL=0
MOVL C01516 V=800.0 PL=0
MOVL C01517 V=800.0 PL=0
MOVL C01518 V=800.0 PL=0
MOVL C01519 V=800.0 PL=0
MOVL C01520 V=800.0 PL=0
MOVL C01521 V=800.0 PL=0
MOVL C01522 V=800.0 PL=0
MOVL C01523 V=800.0 PL=0
MOVL C01524 V=800.0 PL=0
MOVL C01525 V=800.0 PL=0
MOVL C01526 V=800.0 PL=0
MOVL C01527 V=800.0 PL=0
MOVL C01528 V=800.0 PL=0
MOVL C01529 V=800.0 PL=0
MOVL C01530 V=800.0 PL=0
MOVL C01531 V=800.0 PL=0
MOVL C01532 V=800.0 PL=0
MOVL C01533 V=800.0 PL=0
MOVL C01534 V=800.0 PL=0
MOVL C01535 V=800.0 PL=0
MOVL C01536 V=800.0 PL=0
MOVL C01537 V=800.0 PL=0
MOVL C01538 V=800.0 PL=0
MOVL C01539 V=800.0 PL=0
MOVL C01540 V=800.0 PL=0
MOVL C01541 V=800.0 PL=0
MOVL C01542 V=800.0 PL=0
MOVL C01543 V=800.0 PL=0
MOVL C01544 V=800.0 PL=0
MOVL C01545 V=800.0 PL=0
MOVL C01546 V=800.0 PL=0
MOVL C01547 V=800.0 PL=0
MOVL C01548 V=800.0 PL=0
MOVL C01549 V=800.0 PL=0
MOVL C01550 V=800.0 PL=0
MOVL C01551 V=800.0 PL=0
MOVL C01552 V=800.0 PL=0
MOVL C01553 V=800.0 PL=0
MOVL C01554 V=800.0 PL=0
MOVL C01555 V=800.0 PL=0
MOVL C01556 V=800.0 PL=0
MOVL C01557 V=800.0 PL=0
MOVL C01558 V=800.0 PL=0
MOVL C01559 V=800.0 PL=0
MOVL C01560 V=800.0 PL=0
MOVL C01561 V=800.0 PL=0
MOVL C01562 V=800.0 PL=0
MOVL C01563 V=800.0 PL=0
MOVL C01564 V=800.0 PL=0
MOVL C01565 V=800.0 PL=0
MOVL C01566 V=800.0 PL=0
MOVL C01567 V=800.0 PL=0
MOVL C01568 V=800.0 PL=0
MOVL C01569 V=800.0 PL=0
MOVL C01570 V=800.0 PL=0
MOVL C01571 V=800.0 PL=0
MOVL C01572 V=800.0 PL=0
MOVL C01573 V=800.0 PL=0
MOVL C01574 V=800.0 PL=0
MOVL C01575 V=800.0 PL=0
MOVL C01576 V=800.0 PL=0
MOVL C01577 V=800.0 PL=0
MOVL C01578 V=800.0 PL=0
MOVL C01579 V=800.0 PL=0
MOVL C01580 V=800.0 PL=0
MOVL C01581 V=800.0 PL=0
MOVL C01582 V=800.0 PL=0
MOVL C01583 V=800.0 PL=0
MOVL C01584 V=800.0 PL=0
MOVL C01585 V=800.0 PL=0
MOVL C01586 V=800.0 PL=0
MOVL C01587 V=800.0 PL=0
MOVL C01588 V=800.0 PL=0
MOVL C01589 V=800.0 PL=0
MOVL C01590 V=800.0 PL=0
MOVL C01591 V=800.0 PL=0
MOVL C01592 V=800.0 PL=0
MOVL C01593 V=800.0 PL=0
MOVL C01594 V=800.0 PL=0
MOVL C01595 V=800.0 PL=0
MOVL C01596 V=800.0 PL=0
MOVL C01597 V=800.0 PL=0
MOVL C01598 V=800.0 PL=0
MOVL C01599 V=800.0 PL=0
MOVL C01600 V=800.0 PL=0
MOVL C01601 V=800.0 PL=0
MOVL C01602 V=800.0 PL=0
MOVL C01603 V=800.0 PL=0
MOVL C01604 V=800.0 PL=0
MOVL C01605 V=800.0 PL=0
MOVL C01606 V=800.0 PL=0
MOVL C01607 V=800.0 PL=0
MOVL C01608 V=800.0 PL=0
MOVL C01609 V=800.0 PL=0
MOVL C01610 V=800.0 PL=0
MOVL C01611 V=800.0 PL=0
MOVL C01612 V=800.0 PL=0
MOVL C01613 V=800.0 PL=0
MOVL C01614 V=800.0 PL=0
MOVL C01615 V=800.0 PL=0
MOVL C01616 V=800.0 PL=0
MOVL C01617 V=800.0 PL=0
MOVL C01618 V=800.0 PL=0
MOVL C01619 V=800.0 PL=0
MOVL C01620 V=800.0 PL=0
MOVL C01621 V=800.0 PL=0
MOVL C01622 V=800.0 PL=0
MOVL C01623 V=800.0 PL=0
MOVL C01624 V=800.0 PL=0
MOVL C01625 V=800.0 PL=0
MOVL C01626 V=800.0 PL=0
MOVL C01627 V=800.0 PL=0
MOVL C01628 V=800.0 PL=0
MOVL C01629 V=800.0 PL=0
MOVL C01630 V=800.0 PL=0
MOVL C01631 V=800.0 PL=0
MOVL C01632 V=800.0 PL=0
MOVL C01633 V=800.0 PL=0
MOVL C01634 V=800.0 PL=0
MOVL C01635 V=800.0 PL=0
MOVL C01636 V=800.0 PL=0
MOVL C01637 V=800.0 PL=0
MOVL C01638 V=800.0 PL=0
MOVL C01639 V=800.0 PL=0
MOVL C01640 V=800.0 PL=0
MOVL C01641 V=800.0 PL=0
MOVL C01642 V=800.0 PL=0
MOVL C01643 V=800.0 PL=0
MOVL C01644 V=800.0 PL=0
MOVL C01645 V=800.0 PL=0
MOVL C01646 V=800.0 PL=0
MOVL C01647 V=800.0 PL=0
MOVL C01648 V=800.0 PL=0
MOVL C01649 V=800.0 PL=0
MOVL C01650 V=800.0 PL=0
MOVL C01651 V=800.0 PL=0
MOVL C01652 V=800.0 PL=0
MOVL C01653 V=800.0 PL=0
MOVL C01654 V=800.0 PL=0
MOVL C01655 V=800.0 PL=0
MOVL C01656 V=800.0 PL=0
MOVL C01657 V=800.0 PL=0
MOVL C01658 V=800.0 PL=0
MOVL C01659 V=800.0 PL=0
MOVL C01660 V=800.0 PL=0
MOVL C01661 V=800.0 PL=0
MOVL C01662 V=800.0 PL=0
MOVL C01663 V=800.0 PL=0
MOVL C01664 V=800.0 PL=0
MOVL C01665 V=800.0 PL=0
MOVL C01666 V=800.0 PL=0
MOVL C01667 V=800.0 PL=0
MOVL C01668 V=800.0 PL=0
MOVL C01669 V=800.0 PL=0
MOVL C01670 V=800.0 PL=0
MOVL C01671 V=800.0 PL=0
MOVL C01672 V=800.0 PL=0
MOVL C01673 V=800.0 PL=0
MOVL C01674 V=800.0 PL=0
MOVL C01675 V=800.0 PL=0
MOVL C01676 V=800.0 PL=0
MOVL C01677 V=800.0 PL=0
MOVL C01678 V=800.0 PL=0
MOVL C01679 V=800.0 PL=0
MOVL C01680 V=800.0 PL=0
MOVL C01681 V=800.0 PL=0
MOVL C01682 V=800.0 PL=0
MOVL C01683 V=800.0 PL=0
MOVL C01684 V=800.0 PL=0
MOVL C01685 V=800.0 PL=0
MOVL C01686 V=800.0 PL=0
MOVL C01687 V=800.0 PL=0
MOVL C01688 V=800.0 PL=0
MOVL C01689 V=800.0 PL=0
MOVL C01690 V=800.0 PL=0
MOVL C01691 V=800.0 PL=0
MOVL C01692 V=800.0 PL=0
MOVL C01693 V=800.0 PL=0
MOVL C01694 V=800.0 PL=0
MOVL C01695 V=800.0 PL=0
MOVL C01696 V=800.0 PL=0
MOVL C01697 V=800.0 PL=0
MOVL C01698 V=800.0 PL=0
MOVL C01699 V=800.0 PL=0
MOVL C01700 V=800.0 PL=0
MOVL C01701 V=800.0 PL=0
MOVL C01702 V=800.0 PL=0
MOVL C01703 V=800.0 PL=0
MOVL C01704 V=800.0 PL=0
MOVL C01705 V=800.0 PL=0
MOVL C01706 V=800.0 PL=0
MOVL C01707 V=800.0 PL=0
MOVL C01708 V=800.0 PL=0
MOVL C01709 V=800.0 PL=0
MOVL C01710 V=800.0 PL=0
MOVL C01711 V=800.0 PL=0
MOVL C01712 V=800.0 PL=0
MOVL C01713 V=800.0 PL=0
MOVL C01714 V=800.0 PL=0
MOVL C01715 V=800.0 PL=0
MOVL C01716 V=800.0 PL=0
MOVL C01717 V=800.0 PL=0
MOVL C01718 V=800.0 PL=0
MOVL C01719 V=800.0 PL=0
MOVL C01720 V=800.0 PL=0
MOVL C01721 V=800.0 PL=0
MOVL C01722 V=800.0 PL=0
MOVL C01723 V=800.0 PL=0
MOVL C01724 V=800.0 PL=0
MOVL C01725 V=800.0 PL=0
MOVL C01726 V=800.0 PL=0
MOVL C01727 V=800.0 PL=0
MOVL C01728 V=800.0 PL=0
MOVL C01729 V=800.0 PL=0
MOVL C01730 V=800.0 PL=0
MOVL C01731 V=800.0 PL=0
MOVL C01732 V=800.0 PL=0
MOVL C01733 V=800.0 PL=0
MOVL C01734 V=800.0 PL=0
MOVL C01735 V=800.0 PL=0
MOVL C01736 V=800.0 PL=0
MOVL C01737 V=800.0 PL=0
MOVL C01738 V=800.0 PL=0
MOVL C01739 V=800.0 PL=0
MOVL C01740 V=800.0 PL=0
MOVL C01741 V=800.0 PL=0
MOVL C01742 V=800.0 PL=0
MOVL C01743 V=800.0 PL=0
MOVL C01744 V=800.0 PL=0
MOVL C01745 V=800.0 PL=0
MOVL C01746 V=800.0 PL=0
MOVL C01747 V=800.0 PL=0
MOVL C01748 V=800.0 PL=0
MOVL C01749 V=800.0 PL=0
MOVL C01750 V=800.0 PL=0
MOVL C01751 V=800.0 PL=0
MOVL C01752 V=800.0 PL=0
MOVL C01753 V=800.0 PL=0
MOVL C01754 V=800.0 PL=0
MOVL C01755 V=800.0 PL=0
MOVL C01756 V=800.0 PL=0
MOVL C01757 V=800.0 PL=0
MOVL C01758 V=800.0 PL=0
MOVL C01759 V=800.0 PL=0
MOVL C01760 V=800.0 PL=0
MOVL C01761 V=800.0 PL=0
MOVL C01762 V=800.0 PL=0
MOVL C01763 V=800.0 PL=0
MOVL C01764 V=800.0 PL=0
MOVL C01765 V=800.0 PL=0
MOVL C01766 V=800.0 PL=0
MOVL C01767 V=800.0 PL=0
MOVL C01768 V=800.0 PL=0
MOVL C01769 V=800.0 PL=0
MOVL C01770 V=800.0 PL=0
MOVL C01771 V=800.0 PL=0
MOVL C01772 V=800.0 PL=0
MOVL C01773 V=800.0 PL=0
MOVL C01774 V=800.0 PL=0
MOVL C01775 V=800.0 PL=0
MOVL C01776 V=800.0 PL=0
MOVL C01777 V=800.0 PL=0
MOVL C01778 V=800.0 PL=0
MOVL C01779 V=800.0 PL=0
MOVL C01780 V=800.0 PL=0
MOVL C01781 V=800.0 PL=0
MOVL C01782 V=800.0 PL=0
MOVL C01783 V=800.0 PL=0
MOVL C01784 V=800.0 PL=0
MOVL C01785 V=800.0 PL=0
MOVL C01786 V=800.0 PL=0
MOVL C01787 V=800.0 PL=0
MOVL C01788 V=800.0 PL=0
MOVL C01789 V=800.0 PL=0
MOVL C01790 V=800.0 PL=0
MOVL C01791 V=800.0 PL=0
MOVL C01792 V=800.0 PL=0
MOVL C01793 V=800.0 PL=0
MOVL C01794 V=800.0 PL=0
MOVL C01795 V=800.0 PL=0
MOVL C01796 V=800.0 PL=0
MOVL C01797 V=800.0 PL=0
MOVL C01798 V=800.0 PL=0
MOVL C01799 V=800.0 PL=0
MOVL C01800 V=800.0 PL=0
MOVL C01801 V=800.0 PL=0
MOVL C01802 V=800.0 PL=0
MOVL C01803 V=800.0 PL=0
MOVL C01804 V=800.0 PL=0
MOVL C01805 V=800.0 PL=0
MOVL C01806 V=800.0 PL=0
MOVL C01807 V=800.0 PL=0
MOVL C01808 V=800.0 PL=0
MOVL C01809 V=800.0 PL=0
MOVL C01810 V=800.0 PL=0
MOVL C01811 V=800.0 PL=0
MOVL C01812 V=800.0 PL=0
MOVL C01813 V=800.0 PL=0
MOVL C01814 V=800.0 PL=0
MOVL C01815 V=800.0 PL=0
MOVL C01816 V=800.0 PL=0
MOVL C01817 V=800.0 PL=0
MOVL C01818 V=800.0 PL=0
MOVL C01819 V=800.0 PL=0
MOVL C01820 V=800.0 PL=0
MOVL C01821 V=800.0 PL=0
MOVL C01822 V=800.0 PL=0
MOVL C01823 V=800.0 PL=0
MOVL C01824 V=800.0 PL=0
MOVL C01825 V=800.0 PL=0
MOVL C01826 V=800.0 PL=0
MOVL C01827 V=800.0 PL=0
MOVL C01828 V=800.0 PL=0
MOVL C01829 V=800.0 PL=0
MOVL C01830 V=800.0 PL=0
MOVL C01831 V=800.0 PL=0
MOVL C01832 V=800.0 PL=0
MOVL C01833 V=800.0 PL=0
MOVL C01834 V=800.0 PL=0
MOVL C01835 V=800.0 PL=0
MOVL C01836 V=800.0 PL=0
MOVL C01837 V=800.0 PL=0
MOVL C01838 V=800.0 PL=0
MOVL C01839 V=800.0 PL=0
MOVL C01840 V=800.0 PL=0
MOVL C01841 V=800.0 PL=0
MOVL C01842 V=800.0 PL=0
MOVL C01843 V=800.0 PL=0
MOVL C01844 V=800.0 PL=0
MOVL C01845 V=800.0 PL=0
MOVL C01846 V=800.0 PL=0
MOVL C01847 V=800.0 PL=0
MOVL C01848 V=800.0 PL=0
MOVL C01849 V=800.0 PL=0
MOVL C01850 V=800.0 PL=0
MOVL C01851 V=800.0 PL=0
MOVL C01852 V=800.0 PL=0
MOVL C01853 V=800.0 PL=0
MOVL C01854 V=800.0 PL=0
MOVL C01855 V=800.0 PL=0
MOVL C01856 V=800.0 PL=0
MOVL C01857 V=800.0 PL=0
MOVL C01858 V=800.0 PL=0
MOVL C01859 V=800.0 PL=0
MOVL C01860 V=800.0 PL=0
MOVL C01861 V=800.0 PL=0
MOVL C01862 V=800.0 PL=0
MOVL C01863 V=800.0 PL=0
MOVL C01864 V=800.0 PL=0
MOVL C01865 V=800.0 PL=0
MOVL C01866 V=800.0 PL=0
MOVL C01867 V=800.0 PL=0
MOVL C01868 V=800.0 PL=0
MOVL C01869 V=800.0 PL=0
MOVL C01870 V=800.0 PL=0
MOVL C01871 V=800.0 PL=0
MOVL C01872 V=800.0 PL=0
MOVL C01873 V=800.0 PL=0
MOVL C01874 V=800.0 PL=0
MOVL C01875 V=800.0 PL=0
MOVL C01876 V=800.0 PL=0
MOVL C01877 V=800.0 PL=0
MOVL C01878 V=800.0 PL=0
MOVL C01879 V=800.0 PL=0
MOVL C01880 V=800.0 PL=0
MOVL C01881 V=800.0 PL=0
MOVL C01882 V=800.0 PL=0
MOVL C01883 V=800.0 PL=0
MOVL C01884 V=800.0 PL=0
MOVL C01885 V=800.0 PL=0
MOVL C01886 V=800.0 PL=0
MOVL C01887 V=800.0 PL=0
MOVL C01888 V=800.0 PL=0
MOVL C01889 V=800.0 PL=0
MOVL C01890 V=800.0 PL=0
MOVL C01891 V=800.0 PL=0
MOVL C01892 V=800.0 PL=0
MOVL C01893 V=800.0 PL=0
MOVL C01894 V=800.0 PL=0
MOVL C01895 V=800.0 PL=0
MOVL C01896 V=800.0 PL=0
MOVL C01897 V=800.0 PL=0
MOVL C01898 V=800.0 PL=0
MOVL C01899 V=800.0 PL=0
MOVL C01900 V=800.0 PL=0
MOVL C01901 V=800.0 PL=0
MOVL C01902 V=800.0 PL=0
MOVL C01903 V=800.0 PL=0
MOVL C01904 V=800.0 PL=0
MOVL C01905 V=800.0 PL=0
MOVL C01906 V=800.0 PL=0
MOVL C01907 V=800.0 PL=0
MOVL C01908 V=800.0 PL=0
MOVL C01909 V=800.0 PL=0
MOVL C01910 V=800.0 PL=0
MOVL C01911 V=800.0 PL=0
MOVL C01912 V=800.0 PL=0
MOVL C01913 V=800.0 PL=0
MOVL C01914 V=800.0 PL=0
MOVL C01915 V=800.0 PL=0
MOVL C01916 V=800.0 PL=0
MOVL C01917 V=800.0 PL=0
MOVL C01918 V=800.0 PL=0
MOVL C01919 V=800.0 PL=0
MOVL C01920 V=800.0 PL=0
MOVL C01921 V=800.0 PL=0
MOVL C01922 V=800.0 PL=0
MOVL C01923 V=800.0 PL=0
MOVL C01924 V=800.0 PL=0
MOVL C01925 V=800.0 PL=0
MOVL C01926 V=800.0 PL=0
MOVL C01927 V=800.0 PL=0
MOVL C01928 V=800.0 PL=0
MOVL C01929 V=800.0 PL=0
MOVL C01930 V=800.0 PL=0
MOVL C01931 V=800.0 PL=0
MOVL C01932 V=800.0 PL=0
MOVL C01933 V=800.0 PL=0
MOVL C01934 V=800.0 PL=0
MOVL C01935 V=800.0 PL=0
MOVL C01936 V=800.0 PL=0
MOVL C01937 V=800.0 PL=0
MOVL C01938 V=800.0 PL=0
MOVL C01939 V=800.0 PL=0
MOVL C01940 V=800.0 PL=0
MOVL C01941 V=800.0 PL=0
MOVL C01942 V=800.0 PL=0
MOVL C01943 V=800.0 PL=0
MOVL C01944 V=800.0 PL=0
MOVL C01945 V=800.0 PL=0
MOVL C01946 V=800.0 PL=0
MOVL C01947 V=800.0 PL=0
MOVL C01948 V=800.0 PL=0
MOVL C01949 V=800.0 PL=0
MOVL C01950 V=800.0 PL=0
MOVL C01951 V=800.0 PL=0
MOVL C01952 V=800.0 PL=0
MOVL C01953 V=800.0 PL=0
MOVL C01954 V=800.0 PL=0
MOVL C01955 V=800.0 PL=0
MOVL C01956 V=800.0 PL=0
MOVL C01957 V=800.0 PL=0
MOVL C01958 V=800.0 PL=0
MOVL C01959 V=800.0 PL=0
MOVL C01960 V=800.0 PL=0
MOVL C01961 V=800.0 PL=0
MOVL C01962 V=800.0 PL=0
MOVL C01963 V=800.0 PL=0
MOVL C01964 V=800.0 PL=0
MOVL C01965 V=800.0 PL=0
MOVL C01966 V=800.0 PL=0
MOVL C01967 V=800.0 PL=0
MOVL C01968 V=800.0 PL=0
MOVL C01969 V=800.0 PL=0
MOVL C01970 V=800.0 PL=0
MOVL C01971 V=800.0 PL=0
MOVL C01972 V=800.0 PL=0
MOVL C01973 V=800.0 PL=0
MOVL C01974 V=800.0 PL=0
MOVL C01975 V=800.0 PL=0
MOVL C01976 V=800.0 PL=0
MOVL C01977 V=800.0 PL=0
MOVL C01978 V=800.0 PL=0
MOVL C01979 V=800.0 PL=0
MOVL C01980 V=800.0 PL=0
MOVL C01981 V=800.0 PL=0
MOVL C01982 V=800.0 PL=0
MOVL C01983 V=800.0 PL=0
MOVL C01984 V=800.0 PL=0
MOVL C01985 V=800.0 PL=0
MOVL C01986 V=800.0 PL=0
MOVL C01987 V=800.0 PL=0
MOVL C01988 V=800.0 PL=0
MOVL C01989 V=800.0 PL=0
MOVL C01990 V=800.0 PL=0
MOVL C01991 V=800.0 PL=0
MOVL C01992 V=800.0 PL=0
MOVL C01993 V=800.0 PL=0
MOVL C01994 V=800.0 PL=0
MOVL C01995 V=800.0 PL=0
MOVL C01996 V=800.0 PL=0
MOVL C01997 V=800.0 PL=0
MOVL C01998 V=800.0 PL=0
MOVL C01999 V=800.0 PL=0
MOVL C02000 V=800.0 PL=0
MOVL C02001 V=800.0 PL=0
MOVL C02002 V=800.0 PL=0
MOVL C02003 V=800.0 PL=0
MOVL C02004 V=800.0 PL=0
MOVL C02005 V=800.0 PL=0
MOVL C02006 V=800.0 PL=0
MOVL C02007 V=800.0 PL=0
MOVL C02008 V=800.0 PL=0
MOVL C02009 V=800.0 PL=0
MOVL C02010 V=800.0 PL=0
MOVL C02011 V=800.0 PL=0
MOVL C02012 V=800.0 PL=0
MOVL C02013 V=800.0 PL=0
MOVL C02014 V=800.0 PL=0
MOVL C02015 V=800.0 PL=0
MOVL C02016 V=800.0 PL=0
MOVL C02017 V=800.0 PL=0
MOVL C02018 V=800.0 PL=0
MOVL C02019 V=800.0 PL=0
MOVL C02020 V=800.0 PL=0
MOVL C02021 V=800.0 PL=0
MOVL C02022 V=800.0 PL=0
MOVL C02023 V=800.0 PL=0
MOVL C02024 V=800.0 PL=0
MOVL C02025 V=800.0 PL=0
MOVL C02026 V=800.0 PL=0
MOVL C02027 V=800.0 PL=0
MOVL C02028 V=800.0 PL=0
MOVL C02029 V=800.0 PL=0
MOVL C02030 V=800.0 PL=0
MOVL C02031 V=800.0 PL=0
MOVL C02032 V=800.0 PL=0
MOVL C02033 V=800.0 PL=0
MOVL C02034 V=800.0 PL=0
MOVL C02035 V=800.0 PL=0
MOVL C02036 V=800.0 PL=0
MOVL C02037 V=800.0 PL=0
MOVL C02038 V=800.0 PL=0
MOVL C02039 V=800.0 PL=0
MOVL C02040 V=800.0 PL=0
MOVL C02041 V=800.0 PL=0
MOVL C02042 V=800.0 PL=0
MOVL C02043 V=800.0 PL=0
MOVL C02044 V=800.0 PL=0
MOVL C02045 V=800.0 PL=0
MOVL C02046 V=800.0 PL=0
MOVL C02047 V=800.0 PL=0
MOVL C02048 V=800.0 PL=0
MOVL C02049 V=800.0 PL=0
MOVL C02050 V=800.0 PL=0
MOVL C02051 V=800.0 PL=0
MOVL C02052 V=800.0 PL=0
MOVL C02053 V=800.0 PL=0
MOVL C02054 V=800.0 PL=0
MOVL C02055 V=800.0 PL=0
MOVL C02056 V=800.0 PL=0
MOVL C02057 V=800.0 PL=0
MOVL C02058 V=800.0 PL=0
MOVL C02059 V=800.0 PL=0
MOVL C02060 V=800.0 PL=0
MOVL C02061 V=800.0 PL=0
MOVL C02062 V=800.0 PL=0
MOVL C02063 V=800.0 PL=0
MOVL C02064 V=800.0 PL=0
MOVL C02065 V=800.0 PL=0
MOVL C02066 V=800.0 PL=0
MOVL C02067 V=800.0 PL=0
MOVL C02068 V=800.0 PL=0
MOVL C02069 V=800.0 PL=0
MOVL C02070 V=800.0 PL=0
MOVL C02071 V=800.0 PL=0
MOVL C02072 V=800.0 PL=0
MOVL C02073 V=800.0 PL=0
MOVL C02074 V=800.0 PL=0
MOVL C02075 V=800.0 PL=0
MOVL C02076 V=800.0 PL=0
MOVL C02077 V=800.0 PL=0
MOVL C02078 V=800.0 PL=0
MOVL C02079 V=800.0 PL=0
MOVL C02080 V=800.0 PL=0
MOVL C02081 V=800.0 PL=0
MOVL C02082 V=800.0 PL=0
MOVL C02083 V=800.0 PL=0
MOVL C02084 V=800.0 PL=0
MOVL C02085 V=800.0 PL=0
MOVL C02086 V=800.0 PL=0
MOVL C02087 V=800.0 PL=0
MOVL C02088 V=800.0 PL=0
MOVL C02089 V=800.0 PL=0
MOVL C02090 V=800.0 PL=0
MOVL C02091 V=800.0 PL=0
MOVL C02092 V=800.0 PL=0
MOVL C02093 V=800.0 PL=0
MOVL C02094 V=800.0 PL=0
MOVL C02095 V=800.0 PL=0
MOVL C02096 V=800.0 PL=0
MOVL C02097 V=800.0 PL=0
MOVL C02098 V=800.0 PL=0
MOVL C02099 V=800.0 PL=0
MOVL C02100 V=800.0 PL=0
MOVL C02101 V=800.0 PL=0
MOVL C02102 V=800.0 PL=0
MOVL C02103 V=800.0 PL=0
MOVL C02104 V=800.0 PL=0
MOVL C02105 V=800.0 PL=0
MOVL C02106 V=800.0 PL=0
MOVL C02107 V=800.0 PL=0
MOVL C02108 V=800.0 PL=0
MOVL C02109 V=800.0 PL=0
MOVL C02110 V=800.0 PL=0
MOVL C02111 V=800.0 PL=0
MOVL C02112 V=800.0 PL=0
MOVL C02113 V=800.0 PL=0
MOVL C02114 V=800.0 PL=0
MOVL C02115 V=800.0 PL=0
MOVL C02116 V=800.0 PL=0
MOVL C02117 V=800.0 PL=0
MOVL C02118 V=800.0 PL=0
MOVL C02119 V=800.0 PL=0
MOVL C02120 V=800.0 PL=0
MOVL C02121 V=800.0 PL=0
MOVL C02122 V=800.0 PL=0
MOVL C02123 V=800.0 PL=0
MOVL C02124 V=800.0 PL=0
MOVL C02125 V=800.0 PL=0
MOVL C02126 V=800.0 PL=0
MOVL C02127 V=800.0 PL=0
MOVL C02128 V=800.0 PL=0
MOVL C02129 V=800.0 PL=0
MOVL C02130 V=800.0 PL=0
MOVL C02131 V=800.0 PL=0
MOVL C02132 V=800.0 PL=0
MOVL C02133 V=800.0 PL=0
MOVL C02134 V=800.0 PL=0
MOVL C02135 V=800.0 PL=0
MOVL C02136 V=800.0 PL=0
MOVL C02137 V=800.0 PL=0
MOVL C02138 V=800.0 PL=0
MOVL C02139 V=800.0 PL=0
MOVL C02140 V=800.0 PL=0
MOVL C02141 V=800.0 PL=0
MOVL C02142 V=800.0 PL=0
MOVL C02143 V=800.0 PL=0
MOVL C02144 V=800.0 PL=0
MOVL C02145 V=800.0 PL=0
MOVL C02146 V=800.0 PL=0
MOVL C02147 V=800.0 PL=0
MOVL C02148 V=800.0 PL=0
MOVL C02149 V=800.0 PL=0
MOVL C02150 V=800.0 PL=0
MOVL C02151 V=800.0 PL=0
MOVL C02152 V=800.0 PL=0
MOVL C02153 V=800.0 PL=0
MOVL C02154 V=800.0 PL=0
MOVL C02155 V=800.0 PL=0
MOVL C02156 V=800.0 PL=0
MOVL C02157 V=800.0 PL=0
MOVL C02158 V=800.0 PL=0
MOVL C02159 V=800.0 PL=0
MOVL C02160 V=800.0 PL=0
MOVL C02161 V=800.0 PL=0
MOVL C02162 V=800.0 PL=0
MOVL C02163 V=800.0 PL=0
MOVL C02164 V=800.0 PL=0
MOVL C02165 V=800.0 PL=0
MOVL C02166 V=800.0 PL=0
MOVL C02167 V=800.0 PL=0
MOVL C02168 V=800.0 PL=0
MOVL C02169 V=800.0 PL=0
MOVL C02170 V=800.0 PL=0
MOVL C02171 V=800.0 PL=0
MOVL C02172 V=800.0 PL=0
MOVL C02173 V=800.0 PL=0
MOVL C02174 V=800.0 PL=0
MOVL C02175 V=800.0 PL=0
MOVL C02176 V=800.0 PL=0
MOVL C02177 V=800.0 PL=0
MOVL C02178 V=800.0 PL=0
MOVL C02179 V=800.0 PL=0
MOVL C02180 V=800.0 PL=0
MOVL C02181 V=800.0 PL=0
MOVL C02182 V=800.0 PL=0
MOVL C02183 V=800.0 PL=0
